LIN {X 0,Y 646.652,Z 905.532,A -85,B 0,C 180,E1 6708.912,E2 6708.912} C_VEL
LIN {X 0,Y 639.895,Z 980.734,A -85,B 0,C 180,E1 6712.285,E2 6712.285} C_VEL
LIN {X 0,Y 632.591,Z 1048.519,A -85,B 0,C 180,E1 6716.976,E2 6716.976} C_VEL
LIN {X 0,Y 626.439,Z 1105.755,A -85,B 0,C 180,E1 6722.678,E2 6722.678} C_VEL
LIN {X 0,Y 622.279,Z 1152.384,A -85,B 0,C 180,E1 6729.305,E2 6729.305} C_VEL
LIN {X 0,Y 619.924,Z 1184.854,A -85,B 0,C 180,E1 6736.2,E2 6736.2} C_VEL
LIN {X 0,Y 619.217,Z 1203.003,A -85,B 0,C 180,E1 6742.684,E2 6742.684} C_VEL
LIN {X 0,Y 619.285,Z 1209.402,A -85,B 0,C 180,E1 6747.893,E2 6747.893} C_VEL
LIN {X 0,Y 619.07,Z 1206.809,A -85,B 0,C 180,E1 6754.916,E2 6754.916} C_VEL
LIN {X 0,Y 619.272,Z 1193.72,A -85,B 0,C 180,E1 6761.152,E2 6761.152} C_VEL
LIN {X 0,Y 620.479,Z 1169.759,A -85,B 0,C 180,E1 6767.403,E2 6767.403} C_VEL
LIN {X 0,Y 623.213,Z 1133.828,A -85,B 0,C 180,E1 6773.669,E2 6773.669} C_VEL
LIN {X 0,Y 628.639,Z 1081.673,A -85,B 0,C 180,E1 6779.99,E2 6779.99} C_VEL
LIN {X 0,Y 635.999,Z 1018.12,A -85,B 0,C 180,E1 6785.354,E2 6785.354} C_VEL
LIN {X 0,Y 643.399,Z 947.885,A -85,B 0,C 180,E1 6789.377,E2 6789.377} C_VEL
LIN {X 0,Y 649.224,Z 872.681,A -85,B 0,C 180,E1 6792.052,E2 6792.052} C_VEL
LIN {X 0,Y 649.989,Z 821.956,A -85,B 0,C 180,E1 6793.177,E2 6793.177} C_VEL
LIN {X 0,Y 618.006,Z 767.06,A -85,B 0,C 180,E1 6797.097,E2 6797.097} C_VEL
LIN {X 0,Y 618.586,Z 767.06,A -85,B 0,C 180,E1 6805.206,E2 6805.206} C_VEL
LIN {X 0,Y 618.478,Z 767.06,A -85,B 0,C 180,E1 6813.498,E2 6813.498} C_VEL
LIN {X 0,Y 618.567,Z 767.06,A -85,B 0,C 180,E1 6822.165,E2 6822.165} C_VEL
LIN {X 0,Y 618.674,Z 767.06,A -85,B 0,C 180,E1 6830.844,E2 6830.844} C_VEL
LIN {X 0,Y 619.152,Z 767.06,A -85,B 0,C 180,E1 6837.908,E2 6837.908} C_VEL
LIN {X 0,Y 618.57,Z 767.06,A -85,B 0,C 180,E1 6846.859,E2 6846.859} C_VEL
LIN {X 0,Y 618.343,Z 767.06,A -85,B 0,C 180,E1 6854.941,E2 6854.941} C_VEL
LIN {X 0,Y 618.048,Z 767.06,A -85,B 0,C 180,E1 6863.063,E2 6863.063} C_VEL
LIN {X 0,Y 617.959,Z 767.06,A -85,B 0,C 180,E1 6871.87,E2 6871.87} C_VEL
LIN {X 0,Y 617.861,Z 767.06,A -85,B 0,C 180,E1 6880.604,E2 6880.604} C_VEL
LIN {X 0,Y 618.074,Z 767.06,A -85,B 0,C 180,E1 6889.157,E2 6889.157} C_VEL
LIN {X 0,Y 651.016,Z 826.368,A -85,B 0,C 180,E1 6893.12,E2 6893.12} C_VEL
LIN {X 0,Y 646.384,Z 902.657,A -85,B 0,C 180,E1 6895.132,E2 6895.132} C_VEL
LIN {X 0,Y 639.702,Z 974.081,A -85,B 0,C 180,E1 6898.439,E2 6898.439} C_VEL
LIN {X 0,Y 632.109,Z 1042.051,A -85,B 0,C 180,E1 6903.219,E2 6903.219} C_VEL
LIN {X 0,Y 625.727,Z 1100.002,A -85,B 0,C 180,E1 6909.119,E2 6909.119} C_VEL
LIN {X 0,Y 621.471,Z 1145.077,A -85,B 0,C 180,E1 6915.698,E2 6915.698} C_VEL
LIN {X 0,Y 619.614,Z 1173.985,A -85,B 0,C 180,E1 6921.912,E2 6921.912} C_VEL
LIN {X 0,Y 618.989,Z 1191.499,A -85,B 0,C 180,E1 6927.896,E2 6927.896} C_VEL
LIN {X 0,Y 619.03,Z 1199.192,A -85,B 0,C 180,E1 6933.513,E2 6933.513} C_VEL
LIN {X 0,Y 619.006,Z 1198.629,A -85,B 0,C 180,E1 6939.165,E2 6939.165} C_VEL
LIN {X 0,Y 619.22,Z 1187.747,A -85,B 0,C 180,E1 6945.63,E2 6945.63} C_VEL
LIN {X 0,Y 620.1,Z 1164.727,A -85,B 0,C 180,E1 6952.277,E2 6952.277} C_VEL
LIN {X 0,Y 622.657,Z 1130.253,A -85,B 0,C 180,E1 6958.646,E2 6958.646} C_VEL
LIN {X 0,Y 627.586,Z 1081.325,A -85,B 0,C 180,E1 6964.926,E2 6964.926} C_VEL
LIN {X 0,Y 634.691,Z 1018.951,A -85,B 0,C 180,E1 6970.528,E2 6970.528} C_VEL
LIN {X 0,Y 642.172,Z 950.633,A -85,B 0,C 180,E1 6974.718,E2 6974.718} C_VEL
LIN {X 0,Y 648.239,Z 877.127,A -85,B 0,C 180,E1 6977.607,E2 6977.607} C_VEL
LIN {X 0,Y 649.902,Z 822.371,A -85,B 0,C 180,E1 6978.954,E2 6978.954} C_VEL
LIN {X 0,Y 618.301,Z 767.06,A -85,B 0,C 180,E1 6982.858,E2 6982.858} C_VEL
LIN {X 0,Y 618.297,Z 767.06,A -85,B 0,C 180,E1 6991.404,E2 6991.404} C_VEL
LIN {X 0,Y 618.451,Z 767.06,A -85,B 0,C 180,E1 6999.152,E2 6999.152} C_VEL
LIN {X 0,Y 619.304,Z 767.06,A -85,B 0,C 180,E1 7007.969,E2 7007.969} C_VEL
LIN {X 0,Y 619.207,Z 767.06,A -85,B 0,C 180,E1 7017.88,E2 7017.88} C_VEL
LIN {X 0,Y 618.519,Z 767.06,A -85,B 0,C 180,E1 7026.786,E2 7026.786} C_VEL
LIN {X 0,Y 618.33,Z 767.06,A -85,B 0,C 180,E1 7034.912,E2 7034.912} C_VEL
LIN {X 0,Y 618.102,Z 767.06,A -85,B 0,C 180,E1 7043.065,E2 7043.065} C_VEL
LIN {X 0,Y 618.028,Z 767.06,A -85,B 0,C 180,E1 7051.833,E2 7051.833} C_VEL
LIN {X 0,Y 617.735,Z 767.06,A -85,B 0,C 180,E1 7060.577,E2 7060.577} C_VEL
LIN {X 0,Y 618.174,Z 768.815,A -85,B 0,C 180,E1 7063.107,E2 7063.107} C_VEL
LIN {X 0,Y 630.306,Z 788.536,A -85,B 0,C 180,E1 7064.58,E2 7064.58} C_VEL
LIN {X 0,Y 640.035,Z 819.345,A -85,B 0,C 180,E1 7065.934,E2 7065.934} C_VEL
LIN {X 0,Y 645.494,Z 832.84,A -85,B 0,C 180,E1 7066.641,E2 7066.641} C_VEL
LIN {X 0,Y 640.246,Z 910.482,A -85,B 0,C 180,E1 7068.61,E2 7068.61} C_VEL
LIN {X 0,Y 632.996,Z 984.571,A -85,B 0,C 180,E1 7072.046,E2 7072.046} C_VEL
LIN {X 0,Y 625.26,Z 1051.35,A -85,B 0,C 180,E1 7076.795,E2 7076.795} C_VEL
LIN {X 0,Y 618.659,Z 1108.986,A -85,B 0,C 180,E1 7082.705,E2 7082.705} C_VEL
LIN {X 0,Y 614.049,Z 1155.771,A -85,B 0,C 180,E1 7089.619,E2 7089.619} C_VEL
LIN {X 0,Y 611.637,Z 1187.515,A -85,B 0,C 180,E1 7096.74,E2 7096.74} C_VEL
LIN {X 0,Y 610.964,Z 1204.732,A -85,B 0,C 180,E1 7103.585,E2 7103.585} C_VEL
LIN {X 0,Y 610.742,Z 1209.837,A -85,B 0,C 180,E1 7109.287,E2 7109.287} C_VEL
LIN {X 0,Y 610.93,Z 1205.886,A -85,B 0,C 180,E1 7115.696,E2 7115.696} C_VEL
LIN {X 0,Y 611.296,Z 1191.049,A -85,B 0,C 180,E1 7122.171,E2 7122.171} C_VEL
LIN {X 0,Y 612.752,Z 1166.175,A -85,B 0,C 180,E1 7128.391,E2 7128.391} C_VEL
LIN {X 0,Y 616.121,Z 1128.285,A -85,B 0,C 180,E1 7134.768,E2 7134.768} C_VEL
LIN {X 0,Y 622.054,Z 1075.538,A -85,B 0,C 180,E1 7140.989,E2 7140.989} C_VEL
LIN {X 0,Y 629.962,Z 1011.452,A -85,B 0,C 180,E1 7146.255,E2 7146.255} C_VEL
LIN {X 0,Y 637.699,Z 941.735,A -85,B 0,C 180,E1 7150.117,E2 7150.117} C_VEL
LIN {X 0,Y 643.46,Z 869.863,A -85,B 0,C 180,E1 7152.597,E2 7152.597} C_VEL
LIN {X 0,Y 644.183,Z 825.386,A -85,B 0,C 180,E1 7153.602,E2 7153.602} C_VEL
LIN {X 0,Y 610.109,Z 767.06,A -85,B 0,C 180,E1 7157.757,E2 7157.757} C_VEL
LIN {X 0,Y 610.507,Z 767.06,A -85,B 0,C 180,E1 7166.313,E2 7166.313} C_VEL
LIN {X 0,Y 610.224,Z 767.06,A -85,B 0,C 180,E1 7175.097,E2 7175.097} C_VEL
LIN {X 0,Y 610.432,Z 767.06,A -85,B 0,C 180,E1 7183.41,E2 7183.41} C_VEL
LIN {X 0,Y 610.395,Z 767.06,A -85,B 0,C 180,E1 7192.159,E2 7192.159} C_VEL
LIN {X 0,Y 610.543,Z 767.06,A -85,B 0,C 180,E1 7199.302,E2 7199.302} C_VEL
LIN {X 0,Y 610.719,Z 767.06,A -85,B 0,C 180,E1 7206.432,E2 7206.432} C_VEL
LIN {X 0,Y 610.288,Z 767.06,A -85,B 0,C 180,E1 7215.143,E2 7215.143} C_VEL
LIN {X 0,Y 610.126,Z 767.06,A -85,B 0,C 180,E1 7222.681,E2 7222.681} C_VEL
LIN {X 0,Y 610.031,Z 767.06,A -85,B 0,C 180,E1 7230.953,E2 7230.953} C_VEL
LIN {X 0,Y 609.928,Z 767.06,A -85,B 0,C 180,E1 7239.377,E2 7239.377} C_VEL
LIN {X 0,Y 610.104,Z 767.06,A -85,B 0,C 180,E1 7248.363,E2 7248.363} C_VEL
LIN {X 0,Y 644.99,Z 830.304,A -85,B 0,C 180,E1 7252.71,E2 7252.71} C_VEL
LIN {X 0,Y 640.023,Z 905.813,A -85,B 0,C 180,E1 7254.768,E2 7254.768} C_VEL
LIN {X 0,Y 632.651,Z 978.92,A -85,B 0,C 180,E1 7258.259,E2 7258.259} C_VEL
LIN {X 0,Y 624.558,Z 1046.254,A -85,B 0,C 180,E1 7263.167,E2 7263.167} C_VEL
LIN {X 0,Y 617.852,Z 1103.053,A -85,B 0,C 180,E1 7269.154,E2 7269.154} C_VEL
LIN {X 0,Y 613.555,Z 1146.482,A -85,B 0,C 180,E1 7275.693,E2 7275.693} C_VEL
LIN {X 0,Y 611.53,Z 1175.593,A -85,B 0,C 180,E1 7282.163,E2 7282.163} C_VEL
LIN {X 0,Y 610.998,Z 1191.666,A -85,B 0,C 180,E1 7287.868,E2 7287.868} C_VEL
LIN {X 0,Y 611.032,Z 1199.245,A -85,B 0,C 180,E1 7293.559,E2 7293.559} C_VEL
LIN {X 0,Y 610.978,Z 1198.565,A -85,B 0,C 180,E1 7299.286,E2 7299.286} C_VEL
LIN {X 0,Y 611.202,Z 1187.536,A -85,B 0,C 180,E1 7305.84,E2 7305.84} C_VEL
LIN {X 0,Y 612.166,Z 1165.432,A -85,B 0,C 180,E1 7312.328,E2 7312.328} C_VEL
LIN {X 0,Y 614.89,Z 1130.949,A -85,B 0,C 180,E1 7318.838,E2 7318.838} C_VEL
LIN {X 0,Y 620.221,Z 1081.784,A -85,B 0,C 180,E1 7325.251,E2 7325.251} C_VEL
LIN {X 0,Y 627.846,Z 1019.141,A -85,B 0,C 180,E1 7330.943,E2 7330.943} C_VEL
LIN {X 0,Y 635.752,Z 950.839,A -85,B 0,C 180,E1 7335.172,E2 7335.172} C_VEL
LIN {X 0,Y 642.175,Z 877.876,A -85,B 0,C 180,E1 7338.064,E2 7338.064} C_VEL
LIN {X 0,Y 643.929,Z 825.752,A -85,B 0,C 180,E1 7339.389,E2 7339.389} C_VEL
LIN {X 0,Y 610.217,Z 767.06,A -85,B 0,C 180,E1 7343.569,E2 7343.569} C_VEL
LIN {X 0,Y 610.195,Z 767.06,A -85,B 0,C 180,E1 7352.604,E2 7352.604} C_VEL
LIN {X 0,Y 610.314,Z 767.06,A -85,B 0,C 180,E1 7360.38,E2 7360.38} C_VEL
LIN {X 0,Y 611.208,Z 767.06,A -85,B 0,C 180,E1 7369.258,E2 7369.258} C_VEL
LIN {X 0,Y 611.225,Z 767.06,A -85,B 0,C 180,E1 7377.852,E2 7377.852} C_VEL
LIN {X 0,Y 610.649,Z 767.06,A -85,B 0,C 180,E1 7386.404,E2 7386.404} C_VEL
LIN {X 0,Y 610.277,Z 767.06,A -85,B 0,C 180,E1 7395.113,E2 7395.113} C_VEL
LIN {X 0,Y 610.171,Z 767.06,A -85,B 0,C 180,E1 7402.648,E2 7402.648} C_VEL
LIN {X 0,Y 610.093,Z 767.06,A -85,B 0,C 180,E1 7410.955,E2 7410.955} C_VEL
LIN {X 0,Y 609.826,Z 767.06,A -85,B 0,C 180,E1 7419.348,E2 7419.348} C_VEL
LIN {X 0,Y 609.968,Z 768.528,A -85,B 0,C 180,E1 7422.277,E2 7422.277} C_VEL
LIN {X 0,Y 640.035,Z 819.345,A -85,B 0,C 180,E1 7425.934,E2 7425.934} C_VEL
LIN {X 0,Y 641.851,Z 835.895,A -85,B 0,C 180,E1 7426.391,E2 7426.391} C_VEL
LIN {X 0,Y 638.694,Z 854.619,A -85,B 0,C 180,E1 7426.566,E2 7426.566} C_VEL
LIN {X 0,Y 632.966,Z 925.708,A -85,B 0,C 180,E1 7428.72,E2 7428.72} C_VEL
LIN {X 0,Y 624.969,Z 998.18,A -85,B 0,C 180,E1 7432.423,E2 7432.423} C_VEL
LIN {X 0,Y 616.681,Z 1063.626,A -85,B 0,C 180,E1 7437.476,E2 7437.476} C_VEL
LIN {X 0,Y 609.86,Z 1118.897,A -85,B 0,C 180,E1 7443.617,E2 7443.617} C_VEL
LIN {X 0,Y 605.354,Z 1162.455,A -85,B 0,C 180,E1 7450.612,E2 7450.612} C_VEL
LIN {X 0,Y 603.417,Z 1189.883,A -85,B 0,C 180,E1 7457.295,E2 7457.295} C_VEL
LIN {X 0,Y 602.986,Z 1204.729,A -85,B 0,C 180,E1 7463.5,E2 7463.5} C_VEL
LIN {X 0,Y 602.743,Z 1209.837,A -85,B 0,C 180,E1 7469.277,E2 7469.277} C_VEL
LIN {X 0,Y 602.939,Z 1205.886,A -85,B 0,C 180,E1 7475.772,E2 7475.772} C_VEL
LIN {X 0,Y 603.33,Z 1191.046,A -85,B 0,C 180,E1 7482.334,E2 7482.334} C_VEL
LIN {X 0,Y 604.898,Z 1166.177,A -85,B 0,C 180,E1 7488.639,E2 7488.639} C_VEL
LIN {X 0,Y 608.667,Z 1127.165,A -85,B 0,C 180,E1 7495.258,E2 7495.258} C_VEL
LIN {X 0,Y 615.193,Z 1073.255,A -85,B 0,C 180,E1 7501.619,E2 7501.619} C_VEL
LIN {X 0,Y 623.552,Z 1009.569,A -85,B 0,C 180,E1 7506.835,E2 7506.835} C_VEL
LIN {X 0,Y 631.629,Z 940.402,A -85,B 0,C 180,E1 7510.653,E2 7510.653} C_VEL
LIN {X 0,Y 637.635,Z 868.9,A -85,B 0,C 180,E1 7513.108,E2 7513.108} C_VEL
LIN {X 0,Y 638.249,Z 828.483,A -85,B 0,C 180,E1 7514.054,E2 7514.054} C_VEL
LIN {X 0,Y 602.17,Z 767.06,A -85,B 0,C 180,E1 7518.662,E2 7518.662} C_VEL
LIN {X 0,Y 602.419,Z 767.06,A -85,B 0,C 180,E1 7527.485,E2 7527.485} C_VEL
LIN {X 0,Y 602.185,Z 767.06,A -85,B 0,C 180,E1 7535.457,E2 7535.457} C_VEL
LIN {X 0,Y 602.46,Z 767.06,A -85,B 0,C 180,E1 7543.184,E2 7543.184} C_VEL
LIN {X 0,Y 602.432,Z 767.06,A -85,B 0,C 180,E1 7552.054,E2 7552.054} C_VEL
LIN {X 0,Y 602.544,Z 767.06,A -85,B 0,C 180,E1 7559.293,E2 7559.293} C_VEL
LIN {X 0,Y 602.705,Z 767.06,A -85,B 0,C 180,E1 7566.517,E2 7566.517} C_VEL
LIN {X 0,Y 602.244,Z 767.06,A -85,B 0,C 180,E1 7575.35,E2 7575.35} C_VEL
LIN {X 0,Y 602.017,Z 767.06,A -85,B 0,C 180,E1 7583.164,E2 7583.164} C_VEL
LIN {X 0,Y 602.026,Z 767.06,A -85,B 0,C 180,E1 7591.116,E2 7591.116} C_VEL
LIN {X 0,Y 601.862,Z 767.06,A -85,B 0,C 180,E1 7600.01,E2 7600.01} C_VEL
LIN {X 0,Y 602.326,Z 768.684,A -85,B 0,C 180,E1 7607.588,E2 7607.588} C_VEL
LIN {X 0,Y 639.071,Z 831.669,A -85,B 0,C 180,E1 7612.243,E2 7612.243} C_VEL
LIN {X 0,Y 633.792,Z 906.945,A -85,B 0,C 180,E1 7614.327,E2 7614.327} C_VEL
LIN {X 0,Y 626.144,Z 978.79,A -85,B 0,C 180,E1 7617.788,E2 7617.788} C_VEL
LIN {X 0,Y 617.555,Z 1046.251,A -85,B 0,C 180,E1 7622.747,E2 7622.747} C_VEL
LIN {X 0,Y 610.312,Z 1103.709,A -85,B 0,C 180,E1 7628.884,E2 7628.884} C_VEL
LIN {X 0,Y 605.742,Z 1146.922,A -85,B 0,C 180,E1 7635.504,E2 7635.504} C_VEL
LIN {X 0,Y 603.583,Z 1175.885,A -85,B 0,C 180,E1 7642.059,E2 7642.059} C_VEL
LIN {X 0,Y 603.006,Z 1191.828,A -85,B 0,C 180,E1 7647.84,E2 7647.84} C_VEL
LIN {X 0,Y 603.013,Z 1199.293,A -85,B 0,C 180,E1 7653.607,E2 7653.607} C_VEL
LIN {X 0,Y 602.959,Z 1198.499,A -85,B 0,C 180,E1 7659.411,E2 7659.411} C_VEL
LIN {X 0,Y 603.201,Z 1187.324,A -85,B 0,C 180,E1 7666.056,E2 7666.056} C_VEL
LIN {X 0,Y 604.221,Z 1165.961,A -85,B 0,C 180,E1 7672.422,E2 7672.422} C_VEL
LIN {X 0,Y 607.089,Z 1132.198,A -85,B 0,C 180,E1 7678.946,E2 7678.946} C_VEL
LIN {X 0,Y 612.799,Z 1082.461,A -85,B 0,C 180,E1 7685.561,E2 7685.561} C_VEL
LIN {X 0,Y 620.822,Z 1020.755,A -85,B 0,C 180,E1 7691.261,E2 7691.261} C_VEL
LIN {X 0,Y 629.244,Z 952.328,A -85,B 0,C 180,E1 7695.569,E2 7695.569} C_VEL
LIN {X 0,Y 636.186,Z 878.289,A -85,B 0,C 180,E1 7698.538,E2 7698.538} C_VEL
LIN {X 0,Y 637.97,Z 829.221,A -85,B 0,C 180,E1 7699.822,E2 7699.822} C_VEL
LIN {X 0,Y 602.129,Z 767.06,A -85,B 0,C 180,E1 7704.51,E2 7704.51} C_VEL
LIN {X 0,Y 602.148,Z 767.06,A -85,B 0,C 180,E1 7713.39,E2 7713.39} C_VEL
LIN {X 0,Y 602.295,Z 767.06,A -85,B 0,C 180,E1 7721.636,E2 7721.636} C_VEL
LIN {X 0,Y 603.232,Z 767.06,A -85,B 0,C 180,E1 7729.115,E2 7729.115} C_VEL
LIN {X 0,Y 603.222,Z 767.06,A -85,B 0,C 180,E1 7737.824,E2 7737.824} C_VEL
LIN {X 0,Y 602.619,Z 767.06,A -85,B 0,C 180,E1 7746.489,E2 7746.489} C_VEL
LIN {X 0,Y 602.232,Z 767.06,A -85,B 0,C 180,E1 7755.32,E2 7755.32} C_VEL
LIN {X 0,Y 602.087,Z 767.06,A -85,B 0,C 180,E1 7763.169,E2 7763.169} C_VEL
LIN {X 0,Y 602.088,Z 767.06,A -85,B 0,C 180,E1 7771.078,E2 7771.078} C_VEL
LIN {X 0,Y 601.745,Z 767.06,A -85,B 0,C 180,E1 7779.982,E2 7779.982} C_VEL
LIN {X 0,Y 602.006,Z 769.142,A -85,B 0,C 180,E1 7781.44,E2 7781.44} C_VEL
LIN {X 0,Y 638.942,Z 831.754,A -85,B 0,C 180,E1 7786.065,E2 7786.065} C_VEL
LIN {X 0,Y 638.694,Z 854.619,A -85,B 0,C 180,E1 7786.566,E2 7786.566} C_VEL
LIN {X 0,Y 630.175,Z 888.867,A -85,B 0,C 180,E1 7786.933,E2 7786.933} C_VEL
LIN {X 0,Y 622.818,Z 963.473,A -85,B 0,C 180,E1 7789.963,E2 7789.963} C_VEL
LIN {X 0,Y 613.767,Z 1032.869,A -85,B 0,C 180,E1 7794.408,E2 7794.408} C_VEL
LIN {X 0,Y 605.285,Z 1094.461,A -85,B 0,C 180,E1 7800.225,E2 7800.225} C_VEL
LIN {X 0,Y 599.44,Z 1144.557,A -85,B 0,C 180,E1 7807.084,E2 7807.084} C_VEL
LIN {X 0,Y 596.577,Z 1180.801,A -85,B 0,C 180,E1 7814.518,E2 7814.518} C_VEL
LIN {X 0,Y 595.461,Z 1202.16,A -85,B 0,C 180,E1 7821.946,E2 7821.946} C_VEL
LIN {X 0,Y 595.295,Z 1209.402,A -85,B 0,C 180,E1 7827.808,E2 7827.808} C_VEL
LIN {X 0,Y 595.057,Z 1206.8,A -85,B 0,C 180,E1 7835.115,E2 7835.115} C_VEL
LIN {X 0,Y 595.284,Z 1193.106,A -85,B 0,C 180,E1 7841.823,E2 7841.823} C_VEL
LIN {X 0,Y 596.865,Z 1169.068,A -85,B 0,C 180,E1 7848.266,E2 7848.266} C_VEL
LIN {X 0,Y 600.631,Z 1131.177,A -85,B 0,C 180,E1 7855.015,E2 7855.015} C_VEL
LIN {X 0,Y 607.245,Z 1079.171,A -85,B 0,C 180,E1 7861.434,E2 7861.434} C_VEL
LIN {X 0,Y 616.093,Z 1015.607,A -85,B 0,C 180,E1 7866.877,E2 7866.877} C_VEL
LIN {X 0,Y 624.756,Z 946.468,A -85,B 0,C 180,E1 7870.87,E2 7870.87} C_VEL
LIN {X 0,Y 631.517,Z 872.325,A -85,B 0,C 180,E1 7873.527,E2 7873.527} C_VEL
LIN {X 0,Y 632.417,Z 831.751,A -85,B 0,C 180,E1 7874.505,E2 7874.505} C_VEL
LIN {X 0,Y 594.256,Z 767.06,A -85,B 0,C 180,E1 7879.644,E2 7879.644} C_VEL
LIN {X 0,Y 594.349,Z 767.06,A -85,B 0,C 180,E1 7888.727,E2 7888.727} C_VEL
LIN {X 0,Y 594.042,Z 767.06,A -85,B 0,C 180,E1 7896.701,E2 7896.701} C_VEL
LIN {X 0,Y 594.244,Z 767.06,A -85,B 0,C 180,E1 7904.469,E2 7904.469} C_VEL
LIN {X 0,Y 594.437,Z 767.06,A -85,B 0,C 180,E1 7911.947,E2 7911.947} C_VEL
LIN {X 0,Y 594.556,Z 767.06,A -85,B 0,C 180,E1 7919.284,E2 7919.284} C_VEL
LIN {X 0,Y 594.669,Z 767.06,A -85,B 0,C 180,E1 7926.606,E2 7926.606} C_VEL
LIN {X 0,Y 594.204,Z 767.06,A -85,B 0,C 180,E1 7935.563,E2 7935.563} C_VEL
LIN {X 0,Y 593.993,Z 767.06,A -85,B 0,C 180,E1 7943.333,E2 7943.333} C_VEL
LIN {X 0,Y 593.973,Z 767.06,A -85,B 0,C 180,E1 7951.586,E2 7951.586} C_VEL
LIN {X 0,Y 593.795,Z 767.06,A -85,B 0,C 180,E1 7960.667,E2 7960.667} C_VEL
LIN {X 0,Y 594.414,Z 769.008,A -85,B 0,C 180,E1 7966.746,E2 7966.746} C_VEL
LIN {X 0,Y 633.123,Z 835.281,A -85,B 0,C 180,E1 7971.815,E2 7971.815} C_VEL
LIN {X 0,Y 627.447,Z 909.958,A -85,B 0,C 180,E1 7973.955,E2 7973.955} C_VEL
LIN {X 0,Y 619.222,Z 981.916,A -85,B 0,C 180,E1 7977.511,E2 7977.511} C_VEL
LIN {X 0,Y 610.248,Z 1048.399,A -85,B 0,C 180,E1 7982.516,E2 7982.516} C_VEL
LIN {X 0,Y 602.561,Z 1105.875,A -85,B 0,C 180,E1 7988.808,E2 7988.808} C_VEL
LIN {X 0,Y 597.692,Z 1149.281,A -85,B 0,C 180,E1 7995.68,E2 7995.68} C_VEL
LIN {X 0,Y 595.53,Z 1177.485,A -85,B 0,C 180,E1 8002.319,E2 8002.319} C_VEL
LIN {X 0,Y 594.889,Z 1193.365,A -85,B 0,C 180,E1 8008.541,E2 8008.541} C_VEL
LIN {X 0,Y 595.007,Z 1199.34,A -85,B 0,C 180,E1 8013.655,E2 8013.655} C_VEL
LIN {X 0,Y 594.885,Z 1196.995,A -85,B 0,C 180,E1 8020.906,E2 8020.906} C_VEL
LIN {X 0,Y 595.419,Z 1183.037,A -85,B 0,C 180,E1 8027.797,E2 8027.797} C_VEL
LIN {X 0,Y 597.458,Z 1155.363,A -85,B 0,C 180,E1 8035.014,E2 8035.014} C_VEL
LIN {X 0,Y 601.902,Z 1113.172,A -85,B 0,C 180,E1 8042.115,E2 8042.115} C_VEL
LIN {X 0,Y 608.914,Z 1058.814,A -85,B 0,C 180,E1 8048.421,E2 8048.421} C_VEL
LIN {X 0,Y 617.715,Z 993.256,A -85,B 0,C 180,E1 8053.681,E2 8053.681} C_VEL
LIN {X 0,Y 626.349,Z 921.171,A -85,B 0,C 180,E1 8057.505,E2 8057.505} C_VEL
LIN {X 0,Y 632.508,Z 850.17,A -85,B 0,C 180,E1 8059.764,E2 8059.764} C_VEL
LIN {X 0,Y 631.637,Z 831.834,A -85,B 0,C 180,E1 8060.312,E2 8060.312} C_VEL
LIN {X 0,Y 594.082,Z 767.06,A -85,B 0,C 180,E1 8065.523,E2 8065.523} C_VEL
LIN {X 0,Y 594.155,Z 767.06,A -85,B 0,C 180,E1 8073.447,E2 8073.447} C_VEL
LIN {X 0,Y 594.3,Z 767.06,A -85,B 0,C 180,E1 8081.38,E2 8081.38} C_VEL
LIN {X 0,Y 595.216,Z 767.06,A -85,B 0,C 180,E1 8088.966,E2 8088.966} C_VEL
LIN {X 0,Y 595.217,Z 767.06,A -85,B 0,C 180,E1 8097.795,E2 8097.795} C_VEL
LIN {X 0,Y 594.584,Z 767.06,A -85,B 0,C 180,E1 8106.577,E2 8106.577} C_VEL
LIN {X 0,Y 594.191,Z 767.06,A -85,B 0,C 180,E1 8115.533,E2 8115.533} C_VEL
LIN {X 0,Y 594.066,Z 767.06,A -85,B 0,C 180,E1 8123.298,E2 8123.298} C_VEL
LIN {X 0,Y 594.04,Z 767.06,A -85,B 0,C 180,E1 8131.547,E2 8131.547} C_VEL
LIN {X 0,Y 593.742,Z 767.575,A -85,B 0,C 180,E1 8140.469,E2 8140.469} C_VEL
LIN {X 0,Y 633.662,Z 836.021,A -85,B 0,C 180,E1 8145.685,E2 8145.685} C_VEL
LIN {X 0,Y 630.175,Z 888.867,A -85,B 0,C 180,E1 8146.933,E2 8146.933} C_VEL
LIN {X 0,Y 622.012,Z 911.312,A -85,B 0,C 180,E1 8147.149,E2 8147.149} C_VEL
LIN {X 0,Y 613.5,Z 985.783,A -85,B 0,C 180,E1 8150.693,E2 8150.693} C_VEL
LIN {X 0,Y 604.267,Z 1052.795,A -85,B 0,C 180,E1 8155.619,E2 8155.619} C_VEL
LIN {X 0,Y 596.167,Z 1110.284,A -85,B 0,C 180,E1 8161.755,E2 8161.755} C_VEL
LIN {X 0,Y 590.789,Z 1156.571,A -85,B 0,C 180,E1 8168.937,E2 8168.937} C_VEL
LIN {X 0,Y 587.778,Z 1188.725,A -85,B 0,C 180,E1 8176.571,E2 8176.571} C_VEL
LIN {X 0,Y 587.05,Z 1204.724,A -85,B 0,C 180,E1 8183.323,E2 8183.323} C_VEL
LIN {X 0,Y 586.748,Z 1209.837,A -85,B 0,C 180,E1 8189.257,E2 8189.257} C_VEL
LIN {X 0,Y 586.952,Z 1205.919,A -85,B 0,C 180,E1 8195.904,E2 8195.904} C_VEL
LIN {X 0,Y 587.436,Z 1191.04,A -85,B 0,C 180,E1 8202.673,E2 8202.673} C_VEL
LIN {X 0,Y 589.496,Z 1164.51,A -85,B 0,C 180,E1 8209.514,E2 8209.514} C_VEL
LIN {X 0,Y 594.465,Z 1121.523,A -85,B 0,C 180,E1 8216.753,E2 8216.753} C_VEL
LIN {X 0,Y 602.099,Z 1066.601,A -85,B 0,C 180,E1 8223.108,E2 8223.108} C_VEL
LIN {X 0,Y 611.544,Z 1001.134,A -85,B 0,C 180,E1 8228.334,E2 8228.334} C_VEL
LIN {X 0,Y 620.461,Z 929.695,A -85,B 0,C 180,E1 8232.108,E2 8232.108} C_VEL
LIN {X 0,Y 626.59,Z 860.944,A -85,B 0,C 180,E1 8234.299,E2 8234.299} C_VEL
LIN {X 0,Y 626.419,Z 834.814,A -85,B 0,C 180,E1 8234.986,E2 8234.986} C_VEL
LIN {X 0,Y 586.263,Z 767.06,A -85,B 0,C 180,E1 8240.464,E2 8240.464} C_VEL
LIN {X 0,Y 586.296,Z 767.06,A -85,B 0,C 180,E1 8247.987,E2 8247.987} C_VEL
LIN {X 0,Y 586.04,Z 767.06,A -85,B 0,C 180,E1 8256.718,E2 8256.718} C_VEL
LIN {X 0,Y 586.253,Z 767.06,A -85,B 0,C 180,E1 8264.251,E2 8264.251} C_VEL
LIN {X 0,Y 586.452,Z 767.06,A -85,B 0,C 180,E1 8271.836,E2 8271.836} C_VEL
LIN {X 0,Y 586.557,Z 767.06,A -85,B 0,C 180,E1 8279.274,E2 8279.274} C_VEL
LIN {X 0,Y 586.637,Z 767.06,A -85,B 0,C 180,E1 8286.697,E2 8286.697} C_VEL
LIN {X 0,Y 586.454,Z 767.06,A -85,B 0,C 180,E1 8294.239,E2 8294.239} C_VEL
LIN {X 0,Y 585.994,Z 767.06,A -85,B 0,C 180,E1 8303.271,E2 8303.271} C_VEL
LIN {X 0,Y 585.886,Z 767.06,A -85,B 0,C 180,E1 8312.073,E2 8312.073} C_VEL
LIN {X 0,Y 585.798,Z 767.06,A -85,B 0,C 180,E1 8321.342,E2 8321.342} C_VEL
LIN {X 0,Y 586.257,Z 768.601,A -85,B 0,C 180,E1 8325.839,E2 8325.839} C_VEL
LIN {X 0,Y 627.142,Z 837.925,A -85,B 0,C 180,E1 8331.348,E2 8331.348} C_VEL
LIN {X 0,Y 621.227,Z 911.888,A -85,B 0,C 180,E1 8333.531,E2 8333.531} C_VEL
LIN {X 0,Y 612.575,Z 983.23,A -85,B 0,C 180,E1 8337.114,E2 8337.114} C_VEL
LIN {X 0,Y 603.245,Z 1048.719,A -85,B 0,C 180,E1 8342.108,E2 8342.108} C_VEL
LIN {X 0,Y 595.295,Z 1104.999,A -85,B 0,C 180,E1 8348.325,E2 8348.325} C_VEL
LIN {X 0,Y 590.12,Z 1147.905,A -85,B 0,C 180,E1 8355.132,E2 8355.132} C_VEL
LIN {X 0,Y 587.584,Z 1177.753,A -85,B 0,C 180,E1 8362.215,E2 8362.215} C_VEL
LIN {X 0,Y 586.9,Z 1193.501,A -85,B 0,C 180,E1 8368.522,E2 8368.522} C_VEL
LIN {X 0,Y 586.989,Z 1199.387,A -85,B 0,C 180,E1 8373.705,E2 8373.705} C_VEL
LIN {X 0,Y 586.947,Z 1198.365,A -85,B 0,C 180,E1 8379.67,E2 8379.67} C_VEL
LIN {X 0,Y 587.219,Z 1186.952,A -85,B 0,C 180,E1 8386.477,E2 8386.477} C_VEL
LIN {X 0,Y 588.531,Z 1164.891,A -85,B 0,C 180,E1 8393.14,E2 8393.14} C_VEL
LIN {X 0,Y 591.914,Z 1129.776,A -85,B 0,C 180,E1 8399.975,E2 8399.975} C_VEL
LIN {X 0,Y 598.67,Z 1079.518,A -85,B 0,C 180,E1 8406.687,E2 8406.687} C_VEL
LIN {X 0,Y 607.793,Z 1017.294,A -85,B 0,C 180,E1 8412.44,E2 8412.44} C_VEL
LIN {X 0,Y 617.109,Z 949.117,A -85,B 0,C 180,E1 8416.705,E2 8416.705} C_VEL
LIN {X 0,Y 624.477,Z 877.987,A -85,B 0,C 180,E1 8419.545,E2 8419.545} C_VEL
LIN {X 0,Y 626.048,Z 835.954,A -85,B 0,C 180,E1 8420.711,E2 8420.711} C_VEL
LIN {X 0,Y 588.518,Z 772.778,A -85,B 0,C 180,E1 8425.856,E2 8425.856} C_VEL
LIN {X 0,Y 586.079,Z 767.06,A -85,B 0,C 180,E1 8426.456,E2 8426.456} C_VEL
LIN {X 0,Y 586.196,Z 767.06,A -85,B 0,C 180,E1 8434.709,E2 8434.709} C_VEL
LIN {X 0,Y 586.682,Z 767.06,A -85,B 0,C 180,E1 8444.233,E2 8444.233} C_VEL
LIN {X 0,Y 586.54,Z 767.06,A -85,B 0,C 180,E1 8451.808,E2 8451.808} C_VEL
LIN {X 0,Y 586.591,Z 767.06,A -85,B 0,C 180,E1 8459.244,E2 8459.244} C_VEL
LIN {X 0,Y 586.571,Z 767.06,A -85,B 0,C 180,E1 8466.668,E2 8466.668} C_VEL
LIN {X 0,Y 586.457,Z 767.06,A -85,B 0,C 180,E1 8474.209,E2 8474.209} C_VEL
LIN {X 0,Y 586.07,Z 767.06,A -85,B 0,C 180,E1 8483.278,E2 8483.278} C_VEL
LIN {X 0,Y 585.95,Z 767.06,A -85,B 0,C 180,E1 8492.034,E2 8492.034} C_VEL
LIN {X 0,Y 585.991,Z 768.878,A -85,B 0,C 180,E1 8499.556,E2 8499.556} C_VEL
LIN {X 0,Y 622.905,Z 829.875,A -85,B 0,C 180,E1 8504.599,E2 8504.599} C_VEL
LIN {X 0,Y 627.63,Z 844.106,A -85,B 0,C 180,E1 8505.348,E2 8505.348} C_VEL
LIN {X 0,Y 622.012,Z 911.312,A -85,B 0,C 180,E1 8507.149,E2 8507.149} C_VEL
LIN {X 0,Y 612.707,Z 944.277,A -85,B 0,C 180,E1 8508.027,E2 8508.027} C_VEL
LIN {X 0,Y 603.123,Z 1014.101,A -85,B 0,C 180,E1 8512.071,E2 8512.071} C_VEL
LIN {X 0,Y 593.151,Z 1078.693,A -85,B 0,C 180,E1 8517.676,E2 8517.676} C_VEL
LIN {X 0,Y 585.628,Z 1131.143,A -85,B 0,C 180,E1 8524.293,E2 8524.293} C_VEL
LIN {X 0,Y 581.338,Z 1167.92,A -85,B 0,C 180,E1 8530.967,E2 8530.967} C_VEL
LIN {X 0,Y 579.286,Z 1193.288,A -85,B 0,C 180,E1 8537.909,E2 8537.909} C_VEL
LIN {X 0,Y 578.968,Z 1206.789,A -85,B 0,C 180,E1 8544.738,E2 8544.738} C_VEL
LIN {X 0,Y 578.637,Z 1209.838,A -85,B 0,C 180,E1 8550.749,E2 8550.749} C_VEL
LIN {X 0,Y 579.203,Z 1203.517,A -85,B 0,C 180,E1 8557.52,E2 8557.52} C_VEL
LIN {X 0,Y 580.551,Z 1183.675,A -85,B 0,C 180,E1 8565.097,E2 8565.097} C_VEL
LIN {X 0,Y 583.682,Z 1148.476,A -85,B 0,C 180,E1 8572.855,E2 8572.855} C_VEL
LIN {X 0,Y 589.96,Z 1100.701,A -85,B 0,C 180,E1 8579.834,E2 8579.834} C_VEL
LIN {X 0,Y 599.01,Z 1041.871,A -85,B 0,C 180,E1 8585.778,E2 8585.778} C_VEL
LIN {X 0,Y 608.877,Z 973.421,A -85,B 0,C 180,E1 8590.508,E2 8590.508} C_VEL
LIN {X 0,Y 617.236,Z 899.379,A -85,B 0,C 180,E1 8593.774,E2 8593.774} C_VEL
LIN {X 0,Y 620.679,Z 838.301,A -85,B 0,C 180,E1 8595.431,E2 8595.431} C_VEL
LIN {X 0,Y 578.248,Z 767.06,A -85,B 0,C 180,E1 8601.453,E2 8601.453} C_VEL
LIN {X 0,Y 578.248,Z 767.06,A -85,B 0,C 180,E1 8609.252,E2 8609.252} C_VEL
LIN {X 0,Y 578.069,Z 767.06,A -85,B 0,C 180,E1 8618.629,E2 8618.629} C_VEL
LIN {X 0,Y 578.386,Z 767.06,A -85,B 0,C 180,E1 8627.135,E2 8627.135} C_VEL
LIN {X 0,Y 579.023,Z 767.06,A -85,B 0,C 180,E1 8636.26,E2 8636.26} C_VEL
LIN {X 0,Y 579.048,Z 767.06,A -85,B 0,C 180,E1 8645.276,E2 8645.276} C_VEL
LIN {X 0,Y 578.392,Z 767.06,A -85,B 0,C 180,E1 8654.442,E2 8654.442} C_VEL
LIN {X 0,Y 578.065,Z 767.06,A -85,B 0,C 180,E1 8662.38,E2 8662.38} C_VEL
LIN {X 0,Y 577.883,Z 767.06,A -85,B 0,C 180,E1 8671.481,E2 8671.481} C_VEL
LIN {X 0,Y 577.761,Z 767.06,A -85,B 0,C 180,E1 8680.052,E2 8680.052} C_VEL
LIN {X 0,Y 578.298,Z 769.023,A -85,B 0,C 180,E1 8684.937,E2 8684.937} C_VEL
LIN {X 0,Y 620.36,Z 839.379,A -85,B 0,C 180,E1 8690.763,E2 8690.763} C_VEL
LIN {X 0,Y 614.724,Z 917.092,A -85,B 0,C 180,E1 8693.233,E2 8693.233} C_VEL
LIN {X 0,Y 605.555,Z 987.423,A -85,B 0,C 180,E1 8696.894,E2 8696.894} C_VEL
LIN {X 0,Y 595.549,Z 1053.428,A -85,B 0,C 180,E1 8702.105,E2 8702.105} C_VEL
LIN {X 0,Y 587.15,Z 1109.675,A -85,B 0,C 180,E1 8708.58,E2 8708.58} C_VEL
LIN {X 0,Y 581.832,Z 1152.033,A -85,B 0,C 180,E1 8715.666,E2 8715.666} C_VEL
LIN {X 0,Y 579.532,Z 1179.184,A -85,B 0,C 180,E1 8722.484,E2 8722.484} C_VEL
LIN {X 0,Y 578.923,Z 1193.63,A -85,B 0,C 180,E1 8728.501,E2 8728.501} C_VEL
LIN {X 0,Y 578.988,Z 1199.434,A -85,B 0,C 180,E1 8733.757,E2 8733.757} C_VEL
LIN {X 0,Y 578.958,Z 1196.659,A -85,B 0,C 180,E1 8741.331,E2 8741.331} C_VEL
LIN {X 0,Y 579.838,Z 1181.361,A -85,B 0,C 180,E1 8748.688,E2 8748.688} C_VEL
LIN {X 0,Y 582.65,Z 1150.74,A -85,B 0,C 180,E1 8756.479,E2 8756.479} C_VEL
LIN {X 0,Y 587.827,Z 1106.927,A -85,B 0,C 180,E1 8763.689,E2 8763.689} C_VEL
LIN {X 0,Y 596.085,Z 1050.675,A -85,B 0,C 180,E1 8770.059,E2 8770.059} C_VEL
LIN {X 0,Y 605.808,Z 984.65,A -85,B 0,C 180,E1 8775.206,E2 8775.206} C_VEL
LIN {X 0,Y 615.259,Z 910.684,A -85,B 0,C 180,E1 8778.951,E2 8778.951} C_VEL
LIN {X 0,Y 620.213,Z 839.378,A -85,B 0,C 180,E1 8781.162,E2 8781.162} C_VEL
LIN {X 0,Y 584.495,Z 778.715,A -85,B 0,C 180,E1 8786.237,E2 8786.237} C_VEL
LIN {X 0,Y 578.097,Z 767.06,A -85,B 0,C 180,E1 8787.442,E2 8787.442} C_VEL
LIN {X 0,Y 578.264,Z 767.06,A -85,B 0,C 180,E1 8795.993,E2 8795.993} C_VEL
LIN {X 0,Y 578.938,Z 767.06,A -85,B 0,C 180,E1 8805.572,E2 8805.572} C_VEL
LIN {X 0,Y 578.356,Z 767.06,A -85,B 0,C 180,E1 8813.207,E2 8813.207} C_VEL
LIN {X 0,Y 578.615,Z 767.06,A -85,B 0,C 180,E1 8819.234,E2 8819.234} C_VEL
LIN {X 0,Y 578.536,Z 767.06,A -85,B 0,C 180,E1 8826.761,E2 8826.761} C_VEL
LIN {X 0,Y 578.392,Z 767.06,A -85,B 0,C 180,E1 8834.411,E2 8834.411} C_VEL
LIN {X 0,Y 578.159,Z 767.06,A -85,B 0,C 180,E1 8842.344,E2 8842.344} C_VEL
LIN {X 0,Y 577.969,Z 767.06,A -85,B 0,C 180,E1 8851.487,E2 8851.487} C_VEL
LIN {X 0,Y 577.892,Z 768.512,A -85,B 0,C 180,E1 8858.511,E2 8858.511} C_VEL
LIN {X 0,Y 615.856,Z 830.61,A -85,B 0,C 180,E1 8863.949,E2 8863.949} C_VEL
LIN {X 0,Y 621.873,Z 844.951,A -85,B 0,C 180,E1 8864.847,E2 8864.847} C_VEL
LIN {X 0,Y 615.175,Z 921.093,A -85,B 0,C 180,E1 8867.026,E2 8867.026} C_VEL
LIN {X 0,Y 612.707,Z 944.277,A -85,B 0,C 180,E1 8868.027,E2 8868.027} C_VEL
LIN {X 0,Y 602.317,Z 976.103,A -85,B 0,C 180,E1 8869.145,E2 8869.145} C_VEL
LIN {X 0,Y 591.808,Z 1044.155,A -85,B 0,C 180,E1 8873.943,E2 8873.943} C_VEL
LIN {X 0,Y 582.267,Z 1103.279,A -85,B 0,C 180,E1 8880.079,E2 8880.079} C_VEL
LIN {X 0,Y 575.701,Z 1150.853,A -85,B 0,C 180,E1 8887.258,E2 8887.258} C_VEL
LIN {X 0,Y 572.575,Z 1185.315,A -85,B 0,C 180,E1 8895.17,E2 8895.17} C_VEL
LIN {X 0,Y 571.326,Z 1203.507,A -85,B 0,C 180,E1 8902.371,E2 8902.371} C_VEL
LIN {X 0,Y 570.765,Z 1209.837,A -85,B 0,C 180,E1 8909.237,E2 8909.237} C_VEL
LIN {X 0,Y 570.959,Z 1205.886,A -85,B 0,C 180,E1 8916.096,E2 8916.096} C_VEL
LIN {X 0,Y 571.57,Z 1191.034,A -85,B 0,C 180,E1 8923.031,E2 8923.031} C_VEL
LIN {X 0,Y 574.22,Z 1163.028,A -85,B 0,C 180,E1 8930.364,E2 8930.364} C_VEL
LIN {X 0,Y 579.861,Z 1120.319,A -85,B 0,C 180,E1 8937.656,E2 8937.656} C_VEL
LIN {X 0,Y 588.449,Z 1065.276,A -85,B 0,C 180,E1 8944.12,E2 8944.12} C_VEL
LIN {X 0,Y 598.714,Z 1000.505,A -85,B 0,C 180,E1 8949.359,E2 8949.359} C_VEL
LIN {X 0,Y 608.566,Z 928.65,A -85,B 0,C 180,E1 8953.171,E2 8953.171} C_VEL
LIN {X 0,Y 615.189,Z 859.753,A -85,B 0,C 180,E1 8955.374,E2 8955.374} C_VEL
LIN {X 0,Y 614.821,Z 841.717,A -85,B 0,C 180,E1 8955.897,E2 8955.897} C_VEL
LIN {X 0,Y 570.299,Z 767.06,A -85,B 0,C 180,E1 8962.304,E2 8962.304} C_VEL
LIN {X 0,Y 570.24,Z 767.06,A -85,B 0,C 180,E1 8970.538,E2 8970.538} C_VEL
LIN {X 0,Y 570.318,Z 767.06,A -85,B 0,C 180,E1 8980.598,E2 8980.598} C_VEL
LIN {X 0,Y 570.671,Z 767.06,A -85,B 0,C 180,E1 8990.066,E2 8990.066} C_VEL
LIN {X 0,Y 571.155,Z 767.06,A -85,B 0,C 180,E1 8997.732,E2 8997.732} C_VEL
LIN {X 0,Y 570.584,Z 767.06,A -85,B 0,C 180,E1 9006.886,E2 9006.886} C_VEL
LIN {X 0,Y 570.338,Z 767.06,A -85,B 0,C 180,E1 9014.651,E2 9014.651} C_VEL
LIN {X 0,Y 569.912,Z 767.06,A -85,B 0,C 180,E1 9023.371,E2 9023.371} C_VEL
LIN {X 0,Y 569.899,Z 767.06,A -85,B 0,C 180,E1 9031.284,E2 9031.284} C_VEL
LIN {X 0,Y 569.74,Z 767.06,A -85,B 0,C 180,E1 9040.734,E2 9040.734} C_VEL
LIN {X 0,Y 570.079,Z 768.152,A -85,B 0,C 180,E1 9043.942,E2 9043.942} C_VEL
LIN {X 0,Y 614.102,Z 841.665,A -85,B 0,C 180,E1 9050.23,E2 9050.23} C_VEL
LIN {X 0,Y 613.171,Z 873.413,A -85,B 0,C 180,E1 9051.172,E2 9051.172} C_VEL
LIN {X 0,Y 605.124,Z 946.085,A -85,B 0,C 180,E1 9054.024,E2 9054.024} C_VEL
LIN {X 0,Y 594.842,Z 1015.635,A -85,B 0,C 180,E1 9058.39,E2 9058.39} C_VEL
LIN {X 0,Y 584.713,Z 1077.433,A -85,B 0,C 180,E1 9064.147,E2 9064.147} C_VEL
LIN {X 0,Y 577.236,Z 1127.148,A -85,B 0,C 180,E1 9070.831,E2 9070.831} C_VEL
LIN {X 0,Y 573.11,Z 1164.332,A -85,B 0,C 180,E1 9078.149,E2 9078.149} C_VEL
LIN {X 0,Y 571.775,Z 1189.4,A -85,B 0,C 180,E1 9086.2,E2 9086.2} C_VEL
LIN {X 0,Y 570.972,Z 1199.481,A -85,B 0,C 180,E1 9093.809,E2 9093.809} C_VEL
LIN {X 0,Y 570.978,Z 1196.561,A -85,B 0,C 180,E1 9101.492,E2 9101.492} C_VEL
LIN {X 0,Y 571.971,Z 1181.097,A -85,B 0,C 180,E1 9108.955,E2 9108.955} C_VEL
LIN {X 0,Y 574.842,Z 1150.025,A -85,B 0,C 180,E1 9116.919,E2 9116.919} C_VEL
LIN {X 0,Y 580.471,Z 1106.218,A -85,B 0,C 180,E1 9124.175,E2 9124.175} C_VEL
LIN {X 0,Y 589.205,Z 1050.224,A -85,B 0,C 180,E1 9130.561,E2 9130.561} C_VEL
LIN {X 0,Y 599.598,Z 983.619,A -85,B 0,C 180,E1 9135.771,E2 9135.771} C_VEL
LIN {X 0,Y 609.407,Z 909.752,A -85,B 0,C 180,E1 9139.517,E2 9139.517} C_VEL
LIN {X 0,Y 614.396,Z 842.872,A -85,B 0,C 180,E1 9141.621,E2 9141.621} C_VEL
LIN {X 0,Y 580.279,Z 784.159,A -85,B 0,C 180,E1 9146.662,E2 9146.662} C_VEL
LIN {X 0,Y 570.146,Z 767.06,A -85,B 0,C 180,E1 9148.548,E2 9148.548} C_VEL
LIN {X 0,Y 570.327,Z 767.06,A -85,B 0,C 180,E1 9157.3,E2 9157.3} C_VEL
LIN {X 0,Y 571.086,Z 767.06,A -85,B 0,C 180,E1 9166.936,E2 9166.936} C_VEL
LIN {X 0,Y 571.21,Z 767.06,A -85,B 0,C 180,E1 9177.702,E2 9177.702} C_VEL
LIN {X 0,Y 570.522,Z 767.06,A -85,B 0,C 180,E1 9186.856,E2 9186.856} C_VEL
LIN {X 0,Y 570.36,Z 767.06,A -85,B 0,C 180,E1 9194.619,E2 9194.619} C_VEL
LIN {X 0,Y 569.988,Z 767.06,A -85,B 0,C 180,E1 9203.377,E2 9203.377} C_VEL
LIN {X 0,Y 570.002,Z 767.06,A -85,B 0,C 180,E1 9211.242,E2 9211.242} C_VEL
LIN {X 0,Y 569.89,Z 768.339,A -85,B 0,C 180,E1 9217.419,E2 9217.419} C_VEL
LIN {X 0,Y 609.158,Z 831.862,A -85,B 0,C 180,E1 9223.321,E2 9223.321} C_VEL
LIN {X 0,Y 616.019,Z 848.616,A -85,B 0,C 180,E1 9224.395,E2 9224.395} C_VEL
LIN {X 0,Y 608.916,Z 923.92,A -85,B 0,C 180,E1 9226.624,E2 9226.624} C_VEL
LIN {X 0,Y 602.317,Z 976.103,A -85,B 0,C 180,E1 9229.145,E2 9229.145} C_VEL
LIN {X 0,Y 591.388,Z 1006.551,A -85,B 0,C 180,E1 9230.538,E2 9230.538} C_VEL
LIN {X 0,Y 580.607,Z 1070.786,A -85,B 0,C 180,E1 9235.966,E2 9235.966} C_VEL
LIN {X 0,Y 571.581,Z 1125.552,A -85,B 0,C 180,E1 9242.717,E2 9242.717} C_VEL
LIN {X 0,Y 565.953,Z 1166.838,A -85,B 0,C 180,E1 9250.176,E2 9250.176} C_VEL
LIN {X 0,Y 563.421,Z 1193.288,A -85,B 0,C 180,E1 9257.563,E2 9257.563} C_VEL
LIN {X 0,Y 562.981,Z 1206.783,A -85,B 0,C 180,E1 9264.588,E2 9264.588} C_VEL
LIN {X 0,Y 562.644,Z 1209.838,A -85,B 0,C 180,E1 9270.77,E2 9270.77} C_VEL
LIN {X 0,Y 563.258,Z 1203.511,A -85,B 0,C 180,E1 9277.734,E2 9277.734} C_VEL
LIN {X 0,Y 564.743,Z 1183.525,A -85,B 0,C 180,E1 9285.574,E2 9285.574} C_VEL
LIN {X 0,Y 568.196,Z 1149.104,A -85,B 0,C 180,E1 9293.393,E2 9293.393} C_VEL
LIN {X 0,Y 575.171,Z 1102.048,A -85,B 0,C 180,E1 9300.497,E2 9300.497} C_VEL
LIN {X 0,Y 585.523,Z 1042.056,A -85,B 0,C 180,E1 9306.716,E2 9306.716} C_VEL
LIN {X 0,Y 596.185,Z 975.185,A -85,B 0,C 180,E1 9311.423,E2 9311.423} C_VEL
LIN {X 0,Y 605.508,Z 899.895,A -85,B 0,C 180,E1 9314.813,E2 9314.813} C_VEL
LIN {X 0,Y 609.119,Z 845.376,A -85,B 0,C 180,E1 9316.353,E2 9316.353} C_VEL
LIN {X 0,Y 564.01,Z 771.963,A -85,B 0,C 180,E1 9322.838,E2 9322.838} C_VEL
LIN {X 0,Y 562.313,Z 767.06,A -85,B 0,C 180,E1 9323.369,E2 9323.369} C_VEL
LIN {X 0,Y 562.202,Z 767.06,A -85,B 0,C 180,E1 9331.843,E2 9331.843} C_VEL
LIN {X 0,Y 562.333,Z 767.06,A -85,B 0,C 180,E1 9341.945,E2 9341.945} C_VEL
LIN {X 0,Y 562.461,Z 767.06,A -85,B 0,C 180,E1 9351.486,E2 9351.486} C_VEL
LIN {X 0,Y 562.587,Z 767.06,A -85,B 0,C 180,E1 9359.243,E2 9359.243} C_VEL
LIN {X 0,Y 562.554,Z 767.06,A -85,B 0,C 180,E1 9366.985,E2 9366.985} C_VEL
LIN {X 0,Y 562.283,Z 767.06,A -85,B 0,C 180,E1 9374.865,E2 9374.865} C_VEL
LIN {X 0,Y 561.942,Z 767.06,A -85,B 0,C 180,E1 9383.058,E2 9383.058} C_VEL
LIN {X 0,Y 561.824,Z 767.06,A -85,B 0,C 180,E1 9391.786,E2 9391.786} C_VEL
LIN {X 0,Y 561.698,Z 767.06,A -85,B 0,C 180,E1 9399.7,E2 9399.7} C_VEL
LIN {X 0,Y 562.124,Z 769.067,A -85,B 0,C 180,E1 9402.972,E2 9402.972} C_VEL
LIN {X 0,Y 605.899,Z 840.134,A -85,B 0,C 180,E1 9409.387,E2 9409.387} C_VEL
LIN {X 0,Y 609.411,Z 851.687,A -85,B 0,C 180,E1 9410.071,E2 9410.071} C_VEL
LIN {X 0,Y 602.177,Z 923.381,A -85,B 0,C 180,E1 9412.439,E2 9412.439} C_VEL
LIN {X 0,Y 591.954,Z 992.997,A -85,B 0,C 180,E1 9416.252,E2 9416.252} C_VEL
LIN {X 0,Y 580.9,Z 1058.287,A -85,B 0,C 180,E1 9421.657,E2 9421.657} C_VEL
LIN {X 0,Y 571.664,Z 1113.888,A -85,B 0,C 180,E1 9428.409,E2 9428.409} C_VEL
LIN {X 0,Y 566.012,Z 1154.766,A -85,B 0,C 180,E1 9435.653,E2 9435.653} C_VEL
LIN {X 0,Y 563.675,Z 1179.68,A -85,B 0,C 180,E1 9442.272,E2 9442.272} C_VEL
LIN {X 0,Y 562.961,Z 1193.889,A -85,B 0,C 180,E1 9448.459,E2 9448.459} C_VEL
LIN {X 0,Y 562.961,Z 1199.527,A -85,B 0,C 180,E1 9453.864,E2 9453.864} C_VEL
LIN {X 0,Y 563.001,Z 1196.462,A -85,B 0,C 180,E1 9461.657,E2 9461.657} C_VEL
LIN {X 0,Y 564.133,Z 1180.834,A -85,B 0,C 180,E1 9469.228,E2 9469.228} C_VEL
LIN {X 0,Y 567.049,Z 1149.846,A -85,B 0,C 180,E1 9477.258,E2 9477.258} C_VEL
LIN {X 0,Y 573.159,Z 1105.509,A -85,B 0,C 180,E1 9484.672,E2 9484.672} C_VEL
LIN {X 0,Y 582.561,Z 1049.289,A -85,B 0,C 180,E1 9491.115,E2 9491.115} C_VEL
LIN {X 0,Y 593.347,Z 983.385,A -85,B 0,C 180,E1 9496.298,E2 9496.298} C_VEL
LIN {X 0,Y 603.469,Z 910.138,A -85,B 0,C 180,E1 9500.038,E2 9500.038} C_VEL
LIN {X 0,Y 608.784,Z 846.69,A -85,B 0,C 180,E1 9502.062,E2 9502.062} C_VEL
LIN {X 0,Y 575.88,Z 789.148,A -85,B 0,C 180,E1 9507.133,E2 9507.133} C_VEL
LIN {X 0,Y 562.14,Z 767.06,A -85,B 0,C 180,E1 9509.693,E2 9509.693} C_VEL
LIN {X 0,Y 562.258,Z 767.06,A -85,B 0,C 180,E1 9518.625,E2 9518.625} C_VEL
LIN {X 0,Y 563.172,Z 767.06,A -85,B 0,C 180,E1 9528.33,E2 9528.33} C_VEL
LIN {X 0,Y 563.201,Z 767.06,A -85,B 0,C 180,E1 9537.669,E2 9537.669} C_VEL
LIN {X 0,Y 562.49,Z 767.06,A -85,B 0,C 180,E1 9546.954,E2 9546.954} C_VEL
LIN {X 0,Y 562.3,Z 767.06,A -85,B 0,C 180,E1 9554.833,E2 9554.833} C_VEL
LIN {X 0,Y 562.054,Z 767.06,A -85,B 0,C 180,E1 9563.02,E2 9563.02} C_VEL
LIN {X 0,Y 561.907,Z 767.06,A -85,B 0,C 180,E1 9571.772,E2 9571.772} C_VEL
LIN {X 0,Y 562.045,Z 769.071,A -85,B 0,C 180,E1 9576.302,E2 9576.302} C_VEL
LIN {X 0,Y 599.297,Z 827.663,A -85,B 0,C 180,E1 9582.226,E2 9582.226} C_VEL
LIN {X 0,Y 610.137,Z 853.037,A -85,B 0,C 180,E1 9583.947,E2 9583.947} C_VEL
LIN {X 0,Y 602.654,Z 926.746,A -85,B 0,C 180,E1 9586.21,E2 9586.21} C_VEL
LIN {X 0,Y 592.397,Z 999.461,A -85,B 0,C 180,E1 9590.061,E2 9590.061} C_VEL
LIN {X 0,Y 591.388,Z 1006.551,A -85,B 0,C 180,E1 9590.538,E2 9590.538} C_VEL
LIN {X 0,Y 579.966,Z 1035.433,A -85,B 0,C 180,E1 9592.222,E2 9592.222} C_VEL
LIN {X 0,Y 568.806,Z 1096.689,A -85,B 0,C 180,E1 9598.385,E2 9598.385} C_VEL
LIN {X 0,Y 560.95,Z 1144.694,A -85,B 0,C 180,E1 9605.438,E2 9605.438} C_VEL
LIN {X 0,Y 556.814,Z 1179.72,A -85,B 0,C 180,E1 9613.089,E2 9613.089} C_VEL
LIN {X 0,Y 555.517,Z 1200.603,A -85,B 0,C 180,E1 9620.571,E2 9620.571} C_VEL
LIN {X 0,Y 555.285,Z 1209.403,A -85,B 0,C 180,E1 9627.65,E2 9627.65} C_VEL
LIN {X 0,Y 555.049,Z 1206.786,A -85,B 0,C 180,E1 9635.485,E2 9635.485} C_VEL
LIN {X 0,Y 555.543,Z 1193.301,A -85,B 0,C 180,E1 9642.611,E2 9642.611} C_VEL
LIN {X 0,Y 558.149,Z 1166.628,A -85,B 0,C 180,E1 9650.162,E2 9650.162} C_VEL
LIN {X 0,Y 564.197,Z 1124.941,A -85,B 0,C 180,E1 9657.77,E2 9657.77} C_VEL
LIN {X 0,Y 573.516,Z 1071.489,A -85,B 0,C 180,E1 9664.43,E2 9664.43} C_VEL
LIN {X 0,Y 584.738,Z 1008.059,A -85,B 0,C 180,E1 9669.861,E2 9669.861} C_VEL
LIN {X 0,Y 595.698,Z 936.496,A -85,B 0,C 180,E1 9673.899,E2 9673.899} C_VEL
LIN {X 0,Y 603.341,Z 866.933,A -85,B 0,C 180,E1 9676.281,E2 9676.281} C_VEL
LIN {X 0,Y 603.339,Z 848.723,A -85,B 0,C 180,E1 9676.839,E2 9676.839} C_VEL
LIN {X 0,Y 557.309,Z 773.288,A -85,B 0,C 180,E1 9683.667,E2 9683.667} C_VEL
LIN {X 0,Y 554.284,Z 767.06,A -85,B 0,C 180,E1 9684.374,E2 9684.374} C_VEL
LIN {X 0,Y 554.128,Z 767.06,A -85,B 0,C 180,E1 9693.167,E2 9693.167} C_VEL
LIN {X 0,Y 554.287,Z 767.06,A -85,B 0,C 180,E1 9701.673,E2 9701.673} C_VEL
LIN {X 0,Y 554.482,Z 767.06,A -85,B 0,C 180,E1 9711.362,E2 9711.362} C_VEL
LIN {X 0,Y 554.589,Z 767.06,A -85,B 0,C 180,E1 9719.232,E2 9719.232} C_VEL
LIN {X 0,Y 554.548,Z 767.06,A -85,B 0,C 180,E1 9727.086,E2 9727.086} C_VEL
LIN {X 0,Y 554.247,Z 767.06,A -85,B 0,C 180,E1 9735.086,E2 9735.086} C_VEL
LIN {X 0,Y 553.869,Z 767.06,A -85,B 0,C 180,E1 9743.484,E2 9743.484} C_VEL
LIN {X 0,Y 553.747,Z 767.06,A -85,B 0,C 180,E1 9752.305,E2 9752.305} C_VEL
LIN {X 0,Y 553.864,Z 768.483,A -85,B 0,C 180,E1 9761.886,E2 9761.886} C_VEL
LIN {X 0,Y 598.606,Z 840.493,A -85,B 0,C 180,E1 9768.654,E2 9768.654} C_VEL
LIN {X 0,Y 603.614,Z 854.609,A -85,B 0,C 180,E1 9769.597,E2 9769.597} C_VEL
LIN {X 0,Y 596.039,Z 925.328,A -85,B 0,C 180,E1 9771.984,E2 9771.984} C_VEL
LIN {X 0,Y 585.44,Z 994.37,A -85,B 0,C 180,E1 9775.824,E2 9775.824} C_VEL
LIN {X 0,Y 573.679,Z 1060.159,A -85,B 0,C 180,E1 9781.375,E2 9781.375} C_VEL
LIN {X 0,Y 564.141,Z 1114.509,A -85,B 0,C 180,E1 9788.11,E2 9788.11} C_VEL
LIN {X 0,Y 558.193,Z 1155.158,A -85,B 0,C 180,E1 9795.448,E2 9795.448} C_VEL
LIN {X 0,Y 555.619,Z 1181.056,A -85,B 0,C 180,E1 9802.553,E2 9802.553} C_VEL
LIN {X 0,Y 554.783,Z 1195.221,A -85,B 0,C 180,E1 9809.219,E2 9809.219} C_VEL
LIN {X 0,Y 554.812,Z 1199.907,A -85,B 0,C 180,E1 9815.492,E2 9815.492} C_VEL
LIN {X 0,Y 555.349,Z 1194.086,A -85,B 0,C 180,E1 9823.423,E2 9823.423} C_VEL
LIN {X 0,Y 556.565,Z 1175.501,A -85,B 0,C 180,E1 9831.165,E2 9831.165} C_VEL
LIN {X 0,Y 559.755,Z 1142.99,A -85,B 0,C 180,E1 9838.967,E2 9838.967} C_VEL
LIN {X 0,Y 567.043,Z 1097.311,A -85,B 0,C 180,E1 9846.205,E2 9846.205} C_VEL
LIN {X 0,Y 577.506,Z 1038.836,A -85,B 0,C 180,E1 9852.573,E2 9852.573} C_VEL
LIN {X 0,Y 589.019,Z 972.673,A -85,B 0,C 180,E1 9857.473,E2 9857.473} C_VEL
LIN {X 0,Y 599.094,Z 898.317,A -85,B 0,C 180,E1 9861.023,E2 9861.023} C_VEL
LIN {X 0,Y 602.729,Z 849.701,A -85,B 0,C 180,E1 9862.565,E2 9862.565} C_VEL
LIN {X 0,Y 571.012,Z 793.172,A -85,B 0,C 180,E1 9867.702,E2 9867.702} C_VEL
LIN {X 0,Y 554.07,Z 767.06,A -85,B 0,C 180,E1 9870.813,E2 9870.813} C_VEL
LIN {X 0,Y 554.222,Z 767.06,A -85,B 0,C 180,E1 9879.978,E2 9879.978} C_VEL
LIN {X 0,Y 555.14,Z 767.06,A -85,B 0,C 180,E1 9888.159,E2 9888.159} C_VEL
LIN {X 0,Y 555.191,Z 767.06,A -85,B 0,C 180,E1 9897.636,E2 9897.636} C_VEL
LIN {X 0,Y 554.488,Z 767.06,A -85,B 0,C 180,E1 9907.055,E2 9907.055} C_VEL
LIN {X 0,Y 554.255,Z 767.06,A -85,B 0,C 180,E1 9915.053,E2 9915.053} C_VEL
LIN {X 0,Y 553.964,Z 767.06,A -85,B 0,C 180,E1 9923.496,E2 9923.496} C_VEL
LIN {X 0,Y 553.847,Z 767.06,A -85,B 0,C 180,E1 9932.262,E2 9932.262} C_VEL
LIN {X 0,Y 554.031,Z 769.041,A -85,B 0,C 180,E1 9935.07,E2 9935.07} C_VEL
LIN {X 0,Y 591.062,Z 826.072,A -85,B 0,C 180,E1 9941.282,E2 9941.282} C_VEL
LIN {X 0,Y 604.468,Z 855.114,A -85,B 0,C 180,E1 9943.447,E2 9943.447} C_VEL
LIN {X 0,Y 596.558,Z 928.504,A -85,B 0,C 180,E1 9945.744,E2 9945.744} C_VEL
LIN {X 0,Y 585.831,Z 1000.822,A -85,B 0,C 180,E1 9949.638,E2 9949.638} C_VEL
LIN {X 0,Y 579.966,Z 1035.433,A -85,B 0,C 180,E1 9952.222,E2 9952.222} C_VEL
LIN {X 0,Y 568.384,Z 1062.564,A -85,B 0,C 180,E1 9954.196,E2 9954.196} C_VEL
LIN {X 0,Y 558.074,Z 1118.435,A -85,B 0,C 180,E1 9960.88,E2 9960.88} C_VEL
LIN {X 0,Y 551.424,Z 1161.677,A -85,B 0,C 180,E1 9968.462,E2 9968.462} C_VEL
LIN {X 0,Y 547.913,Z 1191.01,A -85,B 0,C 180,E1 9976.391,E2 9976.391} C_VEL
LIN {X 0,Y 547.06,Z 1205.879,A -85,B 0,C 180,E1 9983.632,E2 9983.632} C_VEL
LIN {X 0,Y 546.777,Z 1209.837,A -85,B 0,C 180,E1 9989.203,E2 9989.203} C_VEL
LIN {X 0,Y 547.019,Z 1205.886,A -85,B 0,C 180,E1 9996.364,E2 9996.364} C_VEL
LIN {X 0,Y 548.098,Z 1189.494,A -85,B 0,C 180,E1 10004.143,E2 10004.143} C_VEL
LIN {X 0,Y 551.927,Z 1157.413,A -85,B 0,C 180,E1 10012.444,E2 10012.444} C_VEL
LIN {X 0,Y 559.278,Z 1111.546,A -85,B 0,C 180,E1 10020.105,E2 10020.105} C_VEL
LIN {X 0,Y 569.856,Z 1054.852,A -85,B 0,C 180,E1 10026.562,E2 10026.562} C_VEL
LIN {X 0,Y 581.75,Z 987.827,A -85,B 0,C 180,E1 10031.742,E2 10031.742} C_VEL
LIN {X 0,Y 592.747,Z 913.218,A -85,B 0,C 180,E1 10035.418,E2 10035.418} C_VEL
LIN {X 0,Y 597.543,Z 851.98,A -85,B 0,C 180,E1 10037.342,E2 10037.342} C_VEL
LIN {X 0,Y 553.343,Z 779.442,A -85,B 0,C 180,E1 10044.062,E2 10044.062} C_VEL
LIN {X 0,Y 546.25,Z 767.06,A -85,B 0,C 180,E1 10045.321,E2 10045.321} C_VEL
LIN {X 0,Y 546.022,Z 767.06,A -85,B 0,C 180,E1 10054.512,E2 10054.512} C_VEL
LIN {X 0,Y 546.282,Z 767.06,A -85,B 0,C 180,E1 10063.269,E2 10063.269} C_VEL
LIN {X 0,Y 546.48,Z 767.06,A -85,B 0,C 180,E1 10071.235,E2 10071.235} C_VEL
LIN {X 0,Y 546.603,Z 767.06,A -85,B 0,C 180,E1 10079.221,E2 10079.221} C_VEL
LIN {X 0,Y 546.521,Z 767.06,A -85,B 0,C 180,E1 10087.191,E2 10087.191} C_VEL
LIN {X 0,Y 546.201,Z 767.06,A -85,B 0,C 180,E1 10095.314,E2 10095.314} C_VEL
LIN {X 0,Y 545.848,Z 767.06,A -85,B 0,C 180,E1 10103.78,E2 10103.78} C_VEL
LIN {X 0,Y 545.733,Z 767.06,A -85,B 0,C 180,E1 10112.839,E2 10112.839} C_VEL
LIN {X 0,Y 545.834,Z 768.778,A -85,B 0,C 180,E1 10120.794,E2 10120.794} C_VEL
LIN {X 0,Y 589.404,Z 837.676,A -85,B 0,C 180,E1 10127.607,E2 10127.607} C_VEL
LIN {X 0,Y 597.858,Z 857.382,A -85,B 0,C 180,E1 10129.108,E2 10129.108} C_VEL
LIN {X 0,Y 589.763,Z 928.223,A -85,B 0,C 180,E1 10131.564,E2 10131.564} C_VEL
LIN {X 0,Y 578.672,Z 997.099,A -85,B 0,C 180,E1 10135.482,E2 10135.482} C_VEL
LIN {X 0,Y 566.654,Z 1061.001,A -85,B 0,C 180,E1 10140.987,E2 10140.987} C_VEL
LIN {X 0,Y 556.647,Z 1115.1,A -85,B 0,C 180,E1 10147.8,E2 10147.8} C_VEL
LIN {X 0,Y 550.368,Z 1155.55,A -85,B 0,C 180,E1 10155.236,E2 10155.236} C_VEL
LIN {X 0,Y 547.664,Z 1181.305,A -85,B 0,C 180,E1 10162.445,E2 10162.445} C_VEL
LIN {X 0,Y 546.803,Z 1195.35,A -85,B 0,C 180,E1 10169.208,E2 10169.208} C_VEL
LIN {X 0,Y 546.805,Z 1199.926,A -85,B 0,C 180,E1 10175.573,E2 10175.573} C_VEL
LIN {X 0,Y 547.254,Z 1195.177,A -85,B 0,C 180,E1 10182.81,E2 10182.81} C_VEL
LIN {X 0,Y 548.613,Z 1176.57,A -85,B 0,C 180,E1 10191.062,E2 10191.062} C_VEL
LIN {X 0,Y 551.945,Z 1144.062,A -85,B 0,C 180,E1 10199.099,E2 10199.099} C_VEL
LIN {X 0,Y 559.613,Z 1098.439,A -85,B 0,C 180,E1 10206.49,E2 10206.49} C_VEL
LIN {X 0,Y 570.708,Z 1039.499,A -85,B 0,C 180,E1 10213.015,E2 10213.015} C_VEL
LIN {X 0,Y 582.894,Z 972.749,A -85,B 0,C 180,E1 10218.008,E2 10218.008} C_VEL
LIN {X 0,Y 593.388,Z 898.423,A -85,B 0,C 180,E1 10221.575,E2 10221.575} C_VEL
LIN {X 0,Y 596.971,Z 853.284,A -85,B 0,C 180,E1 10223.034,E2 10223.034} C_VEL
LIN {X 0,Y 567.247,Z 799.238,A -85,B 0,C 180,E1 10228.093,E2 10228.093} C_VEL
LIN {X 0,Y 545.998,Z 767.06,A -85,B 0,C 180,E1 10232.393,E2 10232.393} C_VEL
LIN {X 0,Y 546.232,Z 767.06,A -85,B 0,C 180,E1 10241.36,E2 10241.36} C_VEL
LIN {X 0,Y 546.931,Z 767.06,A -85,B 0,C 180,E1 10249.845,E2 10249.845} C_VEL
LIN {X 0,Y 546.638,Z 767.06,A -85,B 0,C 180,E1 10259.189,E2 10259.189} C_VEL
LIN {X 0,Y 546.457,Z 767.06,A -85,B 0,C 180,E1 10267.16,E2 10267.16} C_VEL
LIN {X 0,Y 546.204,Z 767.06,A -85,B 0,C 180,E1 10275.281,E2 10275.281} C_VEL
LIN {X 0,Y 545.94,Z 767.06,A -85,B 0,C 180,E1 10283.74,E2 10283.74} C_VEL
LIN {X 0,Y 545.822,Z 767.06,A -85,B 0,C 180,E1 10292.795,E2 10292.795} C_VEL
LIN {X 0,Y 546.045,Z 769.109,A -85,B 0,C 180,E1 10293.759,E2 10293.759} C_VEL
LIN {X 0,Y 580.99,Z 821.787,A -85,B 0,C 180,E1 10299.99,E2 10299.99} C_VEL
LIN {X 0,Y 598.576,Z 858.855,A -85,B 0,C 180,E1 10302.977,E2 10302.977} C_VEL
LIN {X 0,Y 590.289,Z 932.643,A -85,B 0,C 180,E1 10305.375,E2 10305.375} C_VEL
LIN {X 0,Y 578.829,Z 1005.17,A -85,B 0,C 180,E1 10309.407,E2 10309.407} C_VEL
LIN {X 0,Y 568.384,Z 1062.564,A -85,B 0,C 180,E1 10314.196,E2 10314.196} C_VEL
LIN {X 0,Y 556.373,Z 1087.862,A -85,B 0,C 180,E1 10316.424,E2 10316.424} C_VEL
LIN {X 0,Y 546.901,Z 1138.67,A -85,B 0,C 180,E1 10323.66,E2 10323.66} C_VEL
LIN {X 0,Y 541.464,Z 1174.679,A -85,B 0,C 180,E1 10331.209,E2 10331.209} C_VEL
LIN {X 0,Y 539.403,Z 1195.277,A -85,B 0,C 180,E1 10337.825,E2 10337.825} C_VEL
LIN {X 0,Y 539.008,Z 1206.774,A -85,B 0,C 180,E1 10344.347,E2 10344.347} C_VEL
LIN {X 0,Y 538.662,Z 1209.838,A -85,B 0,C 180,E1 10350.804,E2 10350.804} C_VEL
LIN {X 0,Y 539.383,Z 1203.503,A -85,B 0,C 180,E1 10358.079,E2 10358.079} C_VEL
LIN {X 0,Y 540.954,Z 1183.523,A -85,B 0,C 180,E1 10366.277,E2 10366.277} C_VEL
LIN {X 0,Y 545.112,Z 1149.178,A -85,B 0,C 180,E1 10374.431,E2 10374.431} C_VEL
LIN {X 0,Y 553.456,Z 1102.446,A -85,B 0,C 180,E1 10381.772,E2 10381.772} C_VEL
LIN {X 0,Y 565.16,Z 1044.205,A -85,B 0,C 180,E1 10388.029,E2 10388.029} C_VEL
LIN {X 0,Y 577.714,Z 975.969,A -85,B 0,C 180,E1 10392.977,E2 10392.977} C_VEL
LIN {X 0,Y 588.368,Z 900.342,A -85,B 0,C 180,E1 10396.457,E2 10396.457} C_VEL
LIN {X 0,Y 591.946,Z 855.649,A -85,B 0,C 180,E1 10397.82,E2 10397.82} C_VEL
LIN {X 0,Y 549.392,Z 785.35,A -85,B 0,C 180,E1 10404.469,E2 10404.469} C_VEL
LIN {X 0,Y 538.148,Z 767.06,A -85,B 0,C 180,E1 10406.677,E2 10406.677} C_VEL
LIN {X 0,Y 537.952,Z 767.06,A -85,B 0,C 180,E1 10416.365,E2 10416.365} C_VEL
LIN {X 0,Y 538.175,Z 767.06,A -85,B 0,C 180,E1 10424.486,E2 10424.486} C_VEL
LIN {X 0,Y 538.308,Z 767.06,A -85,B 0,C 180,E1 10432.731,E2 10432.731} C_VEL
LIN {X 0,Y 538.626,Z 767.06,A -85,B 0,C 180,E1 10439.209,E2 10439.209} C_VEL
LIN {X 0,Y 538.495,Z 767.06,A -85,B 0,C 180,E1 10447.299,E2 10447.299} C_VEL
LIN {X 0,Y 538.176,Z 767.06,A -85,B 0,C 180,E1 10455.548,E2 10455.548} C_VEL
LIN {X 0,Y 537.821,Z 767.06,A -85,B 0,C 180,E1 10464.157,E2 10464.157} C_VEL
LIN {X 0,Y 537.641,Z 767.06,A -85,B 0,C 180,E1 10473.692,E2 10473.692} C_VEL
LIN {X 0,Y 537.796,Z 768.576,A -85,B 0,C 180,E1 10479.63,E2 10479.63} C_VEL
LIN {X 0,Y 580.975,Z 836.323,A -85,B 0,C 180,E1 10486.655,E2 10486.655} C_VEL
LIN {X 0,Y 592.09,Z 860.788,A -85,B 0,C 180,E1 10488.626,E2 10488.626} C_VEL
LIN {X 0,Y 583.581,Z 930.819,A -85,B 0,C 180,E1 10491.124,E2 10491.124} C_VEL
LIN {X 0,Y 571.898,Z 999.695,A -85,B 0,C 180,E1 10495.13,E2 10495.13} C_VEL
LIN {X 0,Y 559.205,Z 1063.91,A -85,B 0,C 180,E1 10500.813,E2 10500.813} C_VEL
LIN {X 0,Y 548.663,Z 1118.233,A -85,B 0,C 180,E1 10507.885,E2 10507.885} C_VEL
LIN {X 0,Y 542.321,Z 1157.691,A -85,B 0,C 180,E1 10515.439,E2 10515.439} C_VEL
LIN {X 0,Y 539.642,Z 1182.681,A -85,B 0,C 180,E1 10522.738,E2 10522.738} C_VEL
LIN {X 0,Y 538.806,Z 1195.477,A -85,B 0,C 180,E1 10529.196,E2 10529.196} C_VEL
LIN {X 0,Y 538.805,Z 1199.944,A -85,B 0,C 180,E1 10535.656,E2 10535.656} C_VEL
LIN {X 0,Y 539.375,Z 1193.809,A -85,B 0,C 180,E1 10543.829,E2 10543.829} C_VEL
LIN {X 0,Y 540.6,Z 1174.871,A -85,B 0,C 180,E1 10551.822,E2 10551.822} C_VEL
LIN {X 0,Y 544.316,Z 1143.673,A -85,B 0,C 180,E1 10559.521,E2 10559.521} C_VEL
LIN {X 0,Y 552.404,Z 1098.27,A -85,B 0,C 180,E1 10566.956,E2 10566.956} C_VEL
LIN {X 0,Y 563.969,Z 1040.146,A -85,B 0,C 180,E1 10573.474,E2 10573.474} C_VEL
LIN {X 0,Y 576.573,Z 974.306,A -85,B 0,C 180,E1 10578.465,E2 10578.465} C_VEL
LIN {X 0,Y 587.395,Z 901.534,A -85,B 0,C 180,E1 10582.03,E2 10582.03} C_VEL
LIN {X 0,Y 591.258,Z 856.768,A -85,B 0,C 180,E1 10583.524,E2 10583.524} C_VEL
LIN {X 0,Y 563.033,Z 804.59,A -85,B 0,C 180,E1 10588.573,E2 10588.573} C_VEL
LIN {X 0,Y 538,Z 767.06,A -85,B 0,C 180,E1 10593.619,E2 10593.619} C_VEL
LIN {X 0,Y 538.364,Z 767.06,A -85,B 0,C 180,E1 10602.775,E2 10602.775} C_VEL
LIN {X 0,Y 538.653,Z 767.06,A -85,B 0,C 180,E1 10611.074,E2 10611.074} C_VEL
LIN {X 0,Y 538.65,Z 767.06,A -85,B 0,C 180,E1 10619.177,E2 10619.177} C_VEL
LIN {X 0,Y 538.428,Z 767.06,A -85,B 0,C 180,E1 10627.267,E2 10627.267} C_VEL
LIN {X 0,Y 538.171,Z 767.06,A -85,B 0,C 180,E1 10635.514,E2 10635.514} C_VEL
LIN {X 0,Y 537.905,Z 767.06,A -85,B 0,C 180,E1 10644.117,E2 10644.117} C_VEL
LIN {X 0,Y 538.027,Z 768.83,A -85,B 0,C 180,E1 10652.337,E2 10652.337} C_VEL
LIN {X 0,Y 572.74,Z 820.623,A -85,B 0,C 180,E1 10658.913,E2 10658.913} C_VEL
LIN {X 0,Y 592.917,Z 861.112,A -85,B 0,C 180,E1 10662.46,E2 10662.46} C_VEL
LIN {X 0,Y 584.123,Z 935.074,A -85,B 0,C 180,E1 10664.93,E2 10664.93} C_VEL
LIN {X 0,Y 572.202,Z 1006.837,A -85,B 0,C 180,E1 10668.996,E2 10668.996} C_VEL
LIN {X 0,Y 559.767,Z 1071.581,A -85,B 0,C 180,E1 10674.612,E2 10674.612} C_VEL
LIN {X 0,Y 556.373,Z 1087.862,A -85,B 0,C 180,E1 10676.424,E2 10676.424} C_VEL
LIN {X 0,Y 544.741,Z 1111.118,A -85,B 0,C 180,E1 10678.938,E2 10678.938} C_VEL
LIN {X 0,Y 536.56,Z 1156.662,A -85,B 0,C 180,E1 10686.707,E2 10686.707} C_VEL
LIN {X 0,Y 532.583,Z 1188.966,A -85,B 0,C 180,E1 10695.245,E2 10695.245} C_VEL
LIN {X 0,Y 531.112,Z 1205.879,A -85,B 0,C 180,E1 10703.44,E2 10703.44} C_VEL
LIN {X 0,Y 530.797,Z 1209.836,A -85,B 0,C 180,E1 10709.179,E2 10709.179} C_VEL
LIN {X 0,Y 531.067,Z 1205.886,A -85,B 0,C 180,E1 10716.556,E2 10716.556} C_VEL
LIN {X 0,Y 532.396,Z 1189.188,A -85,B 0,C 180,E1 10724.68,E2 10724.68} C_VEL
LIN {X 0,Y 536.386,Z 1158.545,A -85,B 0,C 180,E1 10732.875,E2 10732.875} C_VEL
LIN {X 0,Y 544.258,Z 1114.058,A -85,B 0,C 180,E1 10740.626,E2 10740.626} C_VEL
LIN {X 0,Y 555.761,Z 1058.028,A -85,B 0,C 180,E1 10747.256,E2 10747.256} C_VEL
LIN {X 0,Y 568.718,Z 991.751,A -85,B 0,C 180,E1 10752.576,E2 10752.576} C_VEL
LIN {X 0,Y 580.775,Z 917.618,A -85,B 0,C 180,E1 10756.376,E2 10756.376} C_VEL
LIN {X 0,Y 586.035,Z 858.995,A -85,B 0,C 180,E1 10758.327,E2 10758.327} C_VEL
LIN {X 0,Y 545.27,Z 790.922,A -85,B 0,C 180,E1 10764.916,E2 10764.916} C_VEL
LIN {X 0,Y 530.085,Z 767.06,A -85,B 0,C 180,E1 10767.835,E2 10767.835} C_VEL
LIN {X 0,Y 529.925,Z 767.06,A -85,B 0,C 180,E1 10777.286,E2 10777.286} C_VEL
LIN {X 0,Y 530.181,Z 767.06,A -85,B 0,C 180,E1 10785.942,E2 10785.942} C_VEL
LIN {X 0,Y 530.892,Z 767.06,A -85,B 0,C 180,E1 10795.92,E2 10795.92} C_VEL
LIN {X 0,Y 530.854,Z 767.06,A -85,B 0,C 180,E1 10805.756,E2 10805.756} C_VEL
LIN {X 0,Y 530.132,Z 767.06,A -85,B 0,C 180,E1 10815.79,E2 10815.79} C_VEL
LIN {X 0,Y 529.769,Z 767.06,A -85,B 0,C 180,E1 10824.548,E2 10824.548} C_VEL
LIN {X 0,Y 529.643,Z 767.06,A -85,B 0,C 180,E1 10833.97,E2 10833.97} C_VEL
LIN {X 0,Y 529.774,Z 768.685,A -85,B 0,C 180,E1 10838.41,E2 10838.41} C_VEL
LIN {X 0,Y 571.465,Z 833.096,A -85,B 0,C 180,E1 10845.486,E2 10845.486} C_VEL
LIN {X 0,Y 586.379,Z 863.283,A -85,B 0,C 180,E1 10848.112,E2 10848.112} C_VEL
LIN {X 0,Y 577.327,Z 934.138,A -85,B 0,C 180,E1 10850.708,E2 10850.708} C_VEL
LIN {X 0,Y 564.957,Z 1003.334,A -85,B 0,C 180,E1 10854.848,E2 10854.848} C_VEL
LIN {X 0,Y 551.759,Z 1066.793,A -85,B 0,C 180,E1 10860.623,E2 10860.623} C_VEL
LIN {X 0,Y 540.931,Z 1120.067,A -85,B 0,C 180,E1 10867.764,E2 10867.764} C_VEL
LIN {X 0,Y 534.44,Z 1158.477,A -85,B 0,C 180,E1 10875.32,E2 10875.32} C_VEL
LIN {X 0,Y 531.673,Z 1182.927,A -85,B 0,C 180,E1 10882.628,E2 10882.628} C_VEL
LIN {X 0,Y 530.833,Z 1195.599,A -85,B 0,C 180,E1 10889.184,E2 10889.184} C_VEL
LIN {X 0,Y 530.798,Z 1199.963,A -85,B 0,C 180,E1 10895.741,E2 10895.741} C_VEL
LIN {X 0,Y 531.3,Z 1194.901,A -85,B 0,C 180,E1 10903.202,E2 10903.202} C_VEL
LIN {X 0,Y 532.66,Z 1176.553,A -85,B 0,C 180,E1 10911.531,E2 10911.531} C_VEL
LIN {X 0,Y 536.525,Z 1144.827,A -85,B 0,C 180,E1 10919.648,E2 10919.648} C_VEL
LIN {X 0,Y 544.894,Z 1100.105,A -85,B 0,C 180,E1 10927.163,E2 10927.163} C_VEL
LIN {X 0,Y 556.918,Z 1042.601,A -85,B 0,C 180,E1 10933.777,E2 10933.777} C_VEL
LIN {X 0,Y 570.021,Z 977.477,A -85,B 0,C 180,E1 10938.834,E2 10938.834} C_VEL
LIN {X 0,Y 581.594,Z 903.691,A -85,B 0,C 180,E1 10942.534,E2 10942.534} C_VEL
LIN {X 0,Y 585.627,Z 860.12,A -85,B 0,C 180,E1 10944.032,E2 10944.032} C_VEL
LIN {X 0,Y 558.418,Z 809.17,A -85,B 0,C 180,E1 10949.137,E2 10949.137} C_VEL
LIN {X 0,Y 530.035,Z 767.06,A -85,B 0,C 180,E1 10955.202,E2 10955.202} C_VEL
LIN {X 0,Y 530.556,Z 767.06,A -85,B 0,C 180,E1 10964.223,E2 10964.223} C_VEL
LIN {X 0,Y 530.399,Z 767.06,A -85,B 0,C 180,E1 10972.589,E2 10972.589} C_VEL
LIN {X 0,Y 530.672,Z 767.06,A -85,B 0,C 180,E1 10979.165,E2 10979.165} C_VEL
LIN {X 0,Y 530.401,Z 767.06,A -85,B 0,C 180,E1 10987.378,E2 10987.378} C_VEL
LIN {X 0,Y 530.044,Z 767.06,A -85,B 0,C 180,E1 10996.569,E2 10996.569} C_VEL
LIN {X 0,Y 529.823,Z 767.06,A -85,B 0,C 180,E1 11005.627,E2 11005.627} C_VEL
LIN {X 0,Y 530.085,Z 768.944,A -85,B 0,C 180,E1 11010.825,E2 11010.825} C_VEL
LIN {X 0,Y 564.142,Z 818.535,A -85,B 0,C 180,E1 11017.695,E2 11017.695} C_VEL
LIN {X 0,Y 587.362,Z 863.511,A -85,B 0,C 180,E1 11021.936,E2 11021.936} C_VEL
LIN {X 0,Y 578.116,Z 936.711,A -85,B 0,C 180,E1 11024.438,E2 11024.438} C_VEL
LIN {X 0,Y 565.524,Z 1008.911,A -85,B 0,C 180,E1 11028.605,E2 11028.605} C_VEL
LIN {X 0,Y 552.666,Z 1072.688,A -85,B 0,C 180,E1 11034.24,E2 11034.24} C_VEL
LIN {X 0,Y 544.741,Z 1111.118,A -85,B 0,C 180,E1 11038.938,E2 11038.938} C_VEL
LIN {X 0,Y 533.341,Z 1132.179,A -85,B 0,C 180,E1 11041.739,E2 11041.739} C_VEL
LIN {X 0,Y 526.318,Z 1172.173,A -85,B 0,C 180,E1 11049.968,E2 11049.968} C_VEL
LIN {X 0,Y 523.519,Z 1195.271,A -85,B 0,C 180,E1 11057.45,E2 11057.45} C_VEL
LIN {X 0,Y 523.018,Z 1206.768,A -85,B 0,C 180,E1 11064.173,E2 11064.173} C_VEL
LIN {X 0,Y 522.704,Z 1209.837,A -85,B 0,C 180,E1 11070.829,E2 11070.829} C_VEL
LIN {X 0,Y 523.424,Z 1203.497,A -85,B 0,C 180,E1 11078.327,E2 11078.327} C_VEL
LIN {X 0,Y 525.073,Z 1183.521,A -85,B 0,C 180,E1 11086.784,E2 11086.784} C_VEL
LIN {X 0,Y 529.585,Z 1150.858,A -85,B 0,C 180,E1 11094.846,E2 11094.846} C_VEL
LIN {X 0,Y 538.859,Z 1104.283,A -85,B 0,C 180,E1 11102.46,E2 11102.46} C_VEL
LIN {X 0,Y 551.94,Z 1044.605,A -85,B 0,C 180,E1 11109.044,E2 11109.044} C_VEL
LIN {X 0,Y 565.619,Z 976.695,A -85,B 0,C 180,E1 11114.056,E2 11114.056} C_VEL
LIN {X 0,Y 577.019,Z 901.752,A -85,B 0,C 180,E1 11117.557,E2 11117.557} C_VEL
LIN {X 0,Y 580.327,Z 862.798,A -85,B 0,C 180,E1 11118.805,E2 11118.805} C_VEL
LIN {X 0,Y 541.399,Z 796.769,A -85,B 0,C 180,E1 11125.332,E2 11125.332} C_VEL
LIN {X 0,Y 522.044,Z 767.06,A -85,B 0,C 180,E1 11129.208,E2 11129.208} C_VEL
LIN {X 0,Y 521.97,Z 767.06,A -85,B 0,C 180,E1 11138.718,E2 11138.718} C_VEL
LIN {X 0,Y 522.33,Z 767.06,A -85,B 0,C 180,E1 11147.437,E2 11147.437} C_VEL
LIN {X 0,Y 523.136,Z 767.06,A -85,B 0,C 180,E1 11157.524,E2 11157.524} C_VEL
LIN {X 0,Y 522.829,Z 767.06,A -85,B 0,C 180,E1 11165.845,E2 11165.845} C_VEL
LIN {X 0,Y 522.305,Z 767.06,A -85,B 0,C 180,E1 11174.309,E2 11174.309} C_VEL
LIN {X 0,Y 521.76,Z 767.06,A -85,B 0,C 180,E1 11183.726,E2 11183.726} C_VEL
LIN {X 0,Y 521.662,Z 767.06,A -85,B 0,C 180,E1 11192.563,E2 11192.563} C_VEL
LIN {X 0,Y 521.79,Z 768.978,A -85,B 0,C 180,E1 11197.125,E2 11197.125} C_VEL
LIN {X 0,Y 562.835,Z 831.233,A -85,B 0,C 180,E1 11204.408,E2 11204.408} C_VEL
LIN {X 0,Y 580.52,Z 867.452,A -85,B 0,C 180,E1 11207.64,E2 11207.64} C_VEL
LIN {X 0,Y 570.979,Z 938.268,A -85,B 0,C 180,E1 11210.324,E2 11210.324} C_VEL
LIN {X 0,Y 558.299,Z 1005.644,A -85,B 0,C 180,E1 11214.46,E2 11214.46} C_VEL
LIN {X 0,Y 544.627,Z 1068.453,A -85,B 0,C 180,E1 11220.293,E2 11220.293} C_VEL
LIN {X 0,Y 533.205,Z 1121.929,A -85,B 0,C 180,E1 11227.645,E2 11227.645} C_VEL
LIN {X 0,Y 526.374,Z 1160.716,A -85,B 0,C 180,E1 11235.558,E2 11235.558} C_VEL
LIN {X 0,Y 523.614,Z 1185.144,A -85,B 0,C 180,E1 11243.35,E2 11243.35} C_VEL
LIN {X 0,Y 523.149,Z 1197.495,A -85,B 0,C 180,E1 11250.833,E2 11250.833} C_VEL
LIN {X 0,Y 522.889,Z 1198.95,A -85,B 0,C 180,E1 11259.181,E2 11259.181} C_VEL
LIN {X 0,Y 523.428,Z 1188.434,A -85,B 0,C 180,E1 11267.107,E2 11267.107} C_VEL
LIN {X 0,Y 525.622,Z 1166.794,A -85,B 0,C 180,E1 11274.732,E2 11274.732} C_VEL
LIN {X 0,Y 531.644,Z 1130.288,A -85,B 0,C 180,E1 11282.803,E2 11282.803} C_VEL
LIN {X 0,Y 542.333,Z 1079.099,A -85,B 0,C 180,E1 11290.365,E2 11290.365} C_VEL
LIN {X 0,Y 555.592,Z 1018.356,A -85,B 0,C 180,E1 11296.456,E2 11296.456} C_VEL
LIN {X 0,Y 569.267,Z 948.709,A -85,B 0,C 180,E1 11301.062,E2 11301.062} C_VEL
LIN {X 0,Y 579.639,Z 878.707,A -85,B 0,C 180,E1 11303.954,E2 11303.954} C_VEL
LIN {X 0,Y 579.953,Z 863.463,A -85,B 0,C 180,E1 11304.567,E2 11304.567} C_VEL
LIN {X 0,Y 553.212,Z 812.526,A -85,B 0,C 180,E1 11309.832,E2 11309.832} C_VEL
LIN {X 0,Y 523.499,Z 771.623,A -85,B 0,C 180,E1 11316.247,E2 11316.247} C_VEL
LIN {X 0,Y 522.105,Z 767.06,A -85,B 0,C 180,E1 11316.89,E2 11316.89} C_VEL
LIN {X 0,Y 523.013,Z 767.06,A -85,B 0,C 180,E1 11327.42,E2 11327.42} C_VEL
LIN {X 0,Y 523.191,Z 767.06,A -85,B 0,C 180,E1 11337.491,E2 11337.491} C_VEL
LIN {X 0,Y 522.76,Z 767.06,A -85,B 0,C 180,E1 11345.812,E2 11345.812} C_VEL
LIN {X 0,Y 522.296,Z 767.06,A -85,B 0,C 180,E1 11354.274,E2 11354.274} C_VEL
LIN {X 0,Y 521.845,Z 767.06,A -85,B 0,C 180,E1 11363.735,E2 11363.735} C_VEL
LIN {X 0,Y 522.047,Z 768.761,A -85,B 0,C 180,E1 11369.152,E2 11369.152} C_VEL
LIN {X 0,Y 555.692,Z 816.96,A -85,B 0,C 180,E1 11376.43,E2 11376.43} C_VEL
LIN {X 0,Y 581.8,Z 866.131,A -85,B 0,C 180,E1 11381.398,E2 11381.398} C_VEL
LIN {X 0,Y 572.32,Z 937.513,A -85,B 0,C 180,E1 11383.889,E2 11383.889} C_VEL
LIN {X 0,Y 559.1,Z 1009.811,A -85,B 0,C 180,E1 11388.118,E2 11388.118} C_VEL
LIN {X 0,Y 545.737,Z 1073.153,A -85,B 0,C 180,E1 11393.788,E2 11393.788} C_VEL
LIN {X 0,Y 534.767,Z 1125.815,A -85,B 0,C 180,E1 11400.712,E2 11400.712} C_VEL
LIN {X 0,Y 533.341,Z 1132.179,A -85,B 0,C 180,E1 11401.739,E2 11401.739} C_VEL
LIN {X 0,Y 521.965,Z 1150.919,A -85,B 0,C 180,E1 11404.778,E2 11404.778} C_VEL
LIN {X 0,Y 517.055,Z 1183.923,A -85,B 0,C 180,E1 11413.081,E2 11413.081} C_VEL
LIN {X 0,Y 515.508,Z 1203.486,A -85,B 0,C 180,E1 11421.54,E2 11421.54} C_VEL
LIN {X 0,Y 514.799,Z 1209.836,A -85,B 0,C 180,E1 11429.154,E2 11429.154} C_VEL
LIN {X 0,Y 515.095,Z 1205.886,A -85,B 0,C 180,E1 11436.76,E2 11436.76} C_VEL
LIN {X 0,Y 516.728,Z 1188.714,A -85,B 0,C 180,E1 11445.312,E2 11445.312} C_VEL
LIN {X 0,Y 521.099,Z 1157.885,A -85,B 0,C 180,E1 11453.739,E2 11453.739} C_VEL
LIN {X 0,Y 529.927,Z 1113.241,A -85,B 0,C 180,E1 11461.67,E2 11461.67} C_VEL
LIN {X 0,Y 542.675,Z 1057.082,A -85,B 0,C 180,E1 11468.404,E2 11468.404} C_VEL
LIN {X 0,Y 556.661,Z 991.486,A -85,B 0,C 180,E1 11473.731,E2 11473.731} C_VEL
LIN {X 0,Y 569.511,Z 917.398,A -85,B 0,C 180,E1 11477.551,E2 11477.551} C_VEL
LIN {X 0,Y 574.634,Z 866.607,A -85,B 0,C 180,E1 11479.292,E2 11479.292} C_VEL
LIN {X 0,Y 537.923,Z 803.125,A -85,B 0,C 180,E1 11485.689,E2 11485.689} C_VEL
LIN {X 0,Y 513.988,Z 767.06,A -85,B 0,C 180,E1 11490.496,E2 11490.496} C_VEL
LIN {X 0,Y 514.061,Z 767.06,A -85,B 0,C 180,E1 11500.182,E2 11500.182} C_VEL
LIN {X 0,Y 514.48,Z 767.06,A -85,B 0,C 180,E1 11508.969,E2 11508.969} C_VEL
LIN {X 0,Y 515.121,Z 767.06,A -85,B 0,C 180,E1 11517.485,E2 11517.485} C_VEL
LIN {X 0,Y 514.793,Z 767.06,A -85,B 0,C 180,E1 11525.936,E2 11525.936} C_VEL
LIN {X 0,Y 514.249,Z 767.06,A -85,B 0,C 180,E1 11534.538,E2 11534.538} C_VEL
LIN {X 0,Y 513.776,Z 767.06,A -85,B 0,C 180,E1 11543.507,E2 11543.507} C_VEL
LIN {X 0,Y 513.636,Z 767.06,A -85,B 0,C 180,E1 11553.136,E2 11553.136} C_VEL
LIN {X 0,Y 513.756,Z 768.958,A -85,B 0,C 180,E1 11555.74,E2 11555.74} C_VEL
LIN {X 0,Y 554.184,Z 829.37,A -85,B 0,C 180,E1 11563.275,E2 11563.275} C_VEL
LIN {X 0,Y 574.735,Z 870.161,A -85,B 0,C 180,E1 11567.125,E2 11567.125} C_VEL
LIN {X 0,Y 564.715,Z 941.835,A -85,B 0,C 180,E1 11569.908,E2 11569.908} C_VEL
LIN {X 0,Y 551.473,Z 1008.996,A -85,B 0,C 180,E1 11574.143,E2 11574.143} C_VEL
LIN {X 0,Y 536.983,Z 1072.359,A -85,B 0,C 180,E1 11580.207,E2 11580.207} C_VEL
LIN {X 0,Y 525.487,Z 1123.668,A -85,B 0,C 180,E1 11587.5,E2 11587.5} C_VEL
LIN {X 0,Y 518.392,Z 1162.168,A -85,B 0,C 180,E1 11595.605,E2 11595.605} C_VEL
LIN {X 0,Y 515.655,Z 1185.352,A -85,B 0,C 180,E1 11603.247,E2 11603.247} C_VEL
LIN {X 0,Y 515.149,Z 1197.587,A -85,B 0,C 180,E1 11610.846,E2 11610.846} C_VEL
LIN {X 0,Y 514.906,Z 1198.973,A -85,B 0,C 180,E1 11619.189,E2 11619.189} C_VEL
LIN {X 0,Y 515.436,Z 1189.144,A -85,B 0,C 180,E1 11626.918,E2 11626.918} C_VEL
LIN {X 0,Y 517.743,Z 1167.396,A -85,B 0,C 180,E1 11634.854,E2 11634.854} C_VEL
LIN {X 0,Y 524.089,Z 1130.795,A -85,B 0,C 180,E1 11643.123,E2 11643.123} C_VEL
LIN {X 0,Y 535.407,Z 1079.461,A -85,B 0,C 180,E1 11650.835,E2 11650.835} C_VEL
LIN {X 0,Y 549.311,Z 1018.385,A -85,B 0,C 180,E1 11657.022,E2 11657.022} C_VEL
LIN {X 0,Y 563.647,Z 948.629,A -85,B 0,C 180,E1 11661.666,E2 11661.666} C_VEL
LIN {X 0,Y 574.425,Z 878.666,A -85,B 0,C 180,E1 11664.567,E2 11664.567} C_VEL
LIN {X 0,Y 574.22,Z 866.305,A -85,B 0,C 180,E1 11665.148,E2 11665.148} C_VEL
LIN {X 0,Y 548.546,Z 817.095,A -85,B 0,C 180,E1 11670.435,E2 11670.435} C_VEL
LIN {X 0,Y 517.626,Z 773.691,A -85,B 0,C 180,E1 11677.476,E2 11677.476} C_VEL
LIN {X 0,Y 514.149,Z 767.06,A -85,B 0,C 180,E1 11678.795,E2 11678.795} C_VEL
LIN {X 0,Y 514.973,Z 767.06,A -85,B 0,C 180,E1 11688.945,E2 11688.945} C_VEL
LIN {X 0,Y 514.676,Z 767.06,A -85,B 0,C 180,E1 11699.139,E2 11699.139} C_VEL
LIN {X 0,Y 514.37,Z 767.06,A -85,B 0,C 180,E1 11707.609,E2 11707.609} C_VEL
LIN {X 0,Y 514.028,Z 767.06,A -85,B 0,C 180,E1 11716.496,E2 11716.496} C_VEL
LIN {X 0,Y 513.751,Z 767.06,A -85,B 0,C 180,E1 11725.8,E2 11725.8} C_VEL
LIN {X 0,Y 514.086,Z 769.177,A -85,B 0,C 180,E1 11727.351,E2 11727.351} C_VEL
LIN {X 0,Y 543.839,Z 810.298,A -85,B 0,C 180,E1 11734.393,E2 11734.393} C_VEL
LIN {X 0,Y 572.758,Z 861.319,A -85,B 0,C 180,E1 11740.131,E2 11740.131} C_VEL
LIN {X 0,Y 575.974,Z 872.939,A -85,B 0,C 180,E1 11740.963,E2 11740.963} C_VEL
LIN {X 0,Y 565.824,Z 943.082,A -85,B 0,C 180,E1 11743.553,E2 11743.553} C_VEL
LIN {X 0,Y 551.936,Z 1014.514,A -85,B 0,C 180,E1 11747.906,E2 11747.906} C_VEL
LIN {X 0,Y 537.883,Z 1078.11,A -85,B 0,C 180,E1 11753.832,E2 11753.832} C_VEL
LIN {X 0,Y 526.274,Z 1131.126,A -85,B 0,C 180,E1 11761.139,E2 11761.139} C_VEL
LIN {X 0,Y 521.965,Z 1150.919,A -85,B 0,C 180,E1 11764.778,E2 11764.778} C_VEL
LIN {X 0,Y 511.875,Z 1167.289,A -85,B 0,C 180,E1 11768.1,E2 11768.1} C_VEL
LIN {X 0,Y 507.956,Z 1193.914,A -85,B 0,C 180,E1 11776.444,E2 11776.444} C_VEL
LIN {X 0,Y 507.035,Z 1206.763,A -85,B 0,C 180,E1 11783.989,E2 11783.989} C_VEL
LIN {X 0,Y 506.719,Z 1209.837,A -85,B 0,C 180,E1 11790.855,E2 11790.855} C_VEL
LIN {X 0,Y 507.473,Z 1203.491,A -85,B 0,C 180,E1 11798.59,E2 11798.59} C_VEL
LIN {X 0,Y 509.209,Z 1184.079,A -85,B 0,C 180,E1 11807.136,E2 11807.136} C_VEL
LIN {X 0,Y 514.145,Z 1152.377,A -85,B 0,C 180,E1 11815.317,E2 11815.317} C_VEL
LIN {X 0,Y 524.257,Z 1106.239,A -85,B 0,C 180,E1 11823.15,E2 11823.15} C_VEL
LIN {X 0,Y 538.46,Z 1046.95,A -85,B 0,C 180,E1 11829.926,E2 11829.926} C_VEL
LIN {X 0,Y 553.3,Z 979.149,A -85,B 0,C 180,E1 11835.072,E2 11835.072} C_VEL
LIN {X 0,Y 565.732,Z 903.463,A -85,B 0,C 180,E1 11838.678,E2 11838.678} C_VEL
LIN {X 0,Y 568.842,Z 869.938,A -85,B 0,C 180,E1 11839.818,E2 11839.818} C_VEL
LIN {X 0,Y 533.023,Z 807.223,A -85,B 0,C 180,E1 11846.314,E2 11846.314} C_VEL
LIN {X 0,Y 505.975,Z 767.06,A -85,B 0,C 180,E1 11852.141,E2 11852.141} C_VEL
LIN {X 0,Y 506.089,Z 767.06,A -85,B 0,C 180,E1 11861.675,E2 11861.675} C_VEL
LIN {X 0,Y 506.475,Z 767.06,A -85,B 0,C 180,E1 11870.536,E2 11870.536} C_VEL
LIN {X 0,Y 506.67,Z 767.06,A -85,B 0,C 180,E1 11879.159,E2 11879.159} C_VEL
LIN {X 0,Y 506.429,Z 767.06,A -85,B 0,C 180,E1 11887.763,E2 11887.763} C_VEL
LIN {X 0,Y 506.035,Z 767.06,A -85,B 0,C 180,E1 11896.563,E2 11896.563} C_VEL
LIN {X 0,Y 505.724,Z 767.06,A -85,B 0,C 180,E1 11905.799,E2 11905.799} C_VEL
LIN {X 0,Y 505.743,Z 768.941,A -85,B 0,C 180,E1 11914.26,E2 11914.26} C_VEL
LIN {X 0,Y 544.277,Z 825.617,A -85,B 0,C 180,E1 11921.863,E2 11921.863} C_VEL
LIN {X 0,Y 568.848,Z 874.031,A -85,B 0,C 180,E1 11926.638,E2 11926.638} C_VEL
LIN {X 0,Y 558.266,Z 945.786,A -85,B 0,C 180,E1 11929.517,E2 11929.517} C_VEL
LIN {X 0,Y 544.537,Z 1012.779,A -85,B 0,C 180,E1 11933.852,E2 11933.852} C_VEL
LIN {X 0,Y 529.712,Z 1074.62,A -85,B 0,C 180,E1 11939.937,E2 11939.937} C_VEL
LIN {X 0,Y 517.438,Z 1126.709,A -85,B 0,C 180,E1 11947.597,E2 11947.597} C_VEL
LIN {X 0,Y 510.316,Z 1164.145,A -85,B 0,C 180,E1 11955.811,E2 11955.811} C_VEL
LIN {X 0,Y 507.66,Z 1187.452,A -85,B 0,C 180,E1 11964.001,E2 11964.001} C_VEL
LIN {X 0,Y 507.331,Z 1198.911,A -85,B 0,C 180,E1 11972.572,E2 11972.572} C_VEL
LIN {X 0,Y 506.963,Z 1197.516,A -85,B 0,C 180,E1 11981.214,E2 11981.214} C_VEL
LIN {X 0,Y 508.119,Z 1184.782,A -85,B 0,C 180,E1 11989.113,E2 11989.113} C_VEL
LIN {X 0,Y 511.872,Z 1157.518,A -85,B 0,C 180,E1 11997.797,E2 11997.797} C_VEL
LIN {X 0,Y 520.282,Z 1114.955,A -85,B 0,C 180,E1 12006.316,E2 12006.316} C_VEL
LIN {X 0,Y 533.224,Z 1060.725,A -85,B 0,C 180,E1 12013.557,E2 12013.557} C_VEL
LIN {X 0,Y 548.266,Z 995.83,A -85,B 0,C 180,E1 12019.368,E2 12019.368} C_VEL
LIN {X 0,Y 562.589,Z 922.559,A -85,B 0,C 180,E1 12023.58,E2 12023.58} C_VEL
LIN {X 0,Y 569.016,Z 870.727,A -85,B 0,C 180,E1 12025.593,E2 12025.593} C_VEL
LIN {X 0,Y 544.998,Z 823.203,A -85,B 0,C 180,E1 12030.834,E2 12030.834} C_VEL
LIN {X 0,Y 514.787,Z 780.499,A -85,B 0,C 180,E1 12037.915,E2 12037.915} C_VEL
LIN {X 0,Y 506.119,Z 767.06,A -85,B 0,C 180,E1 12040.71,E2 12040.71} C_VEL
LIN {X 0,Y 506.953,Z 767.06,A -85,B 0,C 180,E1 12048.768,E2 12048.768} C_VEL
LIN {X 0,Y 506.679,Z 767.06,A -85,B 0,C 180,E1 12059.125,E2 12059.125} C_VEL
LIN {X 0,Y 506.358,Z 767.06,A -85,B 0,C 180,E1 12067.73,E2 12067.73} C_VEL
LIN {X 0,Y 506.033,Z 767.06,A -85,B 0,C 180,E1 12076.527,E2 12076.527} C_VEL
LIN {X 0,Y 505.945,Z 768.758,A -85,B 0,C 180,E1 12085.272,E2 12085.272} C_VEL
LIN {X 0,Y 535.216,Z 808.406,A -85,B 0,C 180,E1 12092.852,E2 12092.852} C_VEL
LIN {X 0,Y 564.873,Z 859.45,A -85,B 0,C 180,E1 12099.046,E2 12099.046} C_VEL
LIN {X 0,Y 570.61,Z 875.201,A -85,B 0,C 180,E1 12100.401,E2 12100.401} C_VEL
LIN {X 0,Y 559.918,Z 945.42,A -85,B 0,C 180,E1 12103.052,E2 12103.052} C_VEL
LIN {X 0,Y 545.442,Z 1016.138,A -85,B 0,C 180,E1 12107.449,E2 12107.449} C_VEL
LIN {X 0,Y 530.712,Z 1079.782,A -85,B 0,C 180,E1 12113.499,E2 12113.499} C_VEL
LIN {X 0,Y 518.666,Z 1132.409,A -85,B 0,C 180,E1 12120.914,E2 12120.914} C_VEL
LIN {X 0,Y 511.875,Z 1167.289,A -85,B 0,C 180,E1 12128.1,E2 12128.1} C_VEL
LIN {X 0,Y 501.524,Z 1181.163,A -85,B 0,C 180,E1 12131.606,E2 12131.606} C_VEL
LIN {X 0,Y 499.551,Z 1202.149,A -85,B 0,C 180,E1 12140.386,E2 12140.386} C_VEL
LIN {X 0,Y 499.297,Z 1209.395,A -85,B 0,C 180,E1 12147.386,E2 12147.386} C_VEL
LIN {X 0,Y 499.24,Z 1208.366,A -85,B 0,C 180,E1 12154.353,E2 12154.353} C_VEL
LIN {X 0,Y 499.616,Z 1197.202,A -85,B 0,C 180,E1 12162.264,E2 12162.264} C_VEL
LIN {X 0,Y 502.545,Z 1174.69,A -85,B 0,C 180,E1 12170.302,E2 12170.302} C_VEL
LIN {X 0,Y 510.015,Z 1137.069,A -85,B 0,C 180,E1 12178.709,E2 12178.709} C_VEL
LIN {X 0,Y 522.724,Z 1084.509,A -85,B 0,C 180,E1 12186.49,E2 12186.49} C_VEL
LIN {X 0,Y 537.997,Z 1022.313,A -85,B 0,C 180,E1 12192.65,E2 12192.65} C_VEL
LIN {X 0,Y 552.598,Z 953.245,A -85,B 0,C 180,E1 12197.106,E2 12197.106} C_VEL
LIN {X 0,Y 563.332,Z 882.565,A -85,B 0,C 180,E1 12199.924,E2 12199.924} C_VEL
LIN {X 0,Y 562.537,Z 872.525,A -85,B 0,C 180,E1 12200.445,E2 12200.445} C_VEL
LIN {X 0,Y 528.173,Z 811.434,A -85,B 0,C 180,E1 12206.95,E2 12206.95} C_VEL
LIN {X 0,Y 497.905,Z 767.06,A -85,B 0,C 180,E1 12213.805,E2 12213.805} C_VEL
LIN {X 0,Y 498.122,Z 767.06,A -85,B 0,C 180,E1 12223.521,E2 12223.521} C_VEL
LIN {X 0,Y 498.329,Z 767.06,A -85,B 0,C 180,E1 12232.145,E2 12232.145} C_VEL
LIN {X 0,Y 498.672,Z 767.06,A -85,B 0,C 180,E1 12239.146,E2 12239.146} C_VEL
LIN {X 0,Y 498.408,Z 767.06,A -85,B 0,C 180,E1 12247.889,E2 12247.889} C_VEL
LIN {X 0,Y 498.011,Z 767.06,A -85,B 0,C 180,E1 12256.838,E2 12256.838} C_VEL
LIN {X 0,Y 497.694,Z 767.06,A -85,B 0,C 180,E1 12266.246,E2 12266.246} C_VEL
LIN {X 0,Y 497.703,Z 768.782,A -85,B 0,C 180,E1 12272.656,E2 12272.656} C_VEL
LIN {X 0,Y 534.85,Z 822.679,A -85,B 0,C 180,E1 12280.467,E2 12280.467} C_VEL
LIN {X 0,Y 563.186,Z 876.467,A -85,B 0,C 180,E1 12286.101,E2 12286.101} C_VEL
LIN {X 0,Y 552.054,Z 948.527,A -85,B 0,C 180,E1 12289.059,E2 12289.059} C_VEL
LIN {X 0,Y 537.868,Z 1015.006,A -85,B 0,C 180,E1 12293.446,E2 12293.446} C_VEL
LIN {X 0,Y 522.74,Z 1075.465,A -85,B 0,C 180,E1 12299.494,E2 12299.494} C_VEL
LIN {X 0,Y 510.255,Z 1126.289,A -85,B 0,C 180,E1 12307.059,E2 12307.059} C_VEL
LIN {X 0,Y 502.504,Z 1164.481,A -85,B 0,C 180,E1 12315.586,E2 12315.586} C_VEL
LIN {X 0,Y 499.709,Z 1185.769,A -85,B 0,C 180,E1 12323.03,E2 12323.03} C_VEL
LIN {X 0,Y 499.161,Z 1197.769,A -85,B 0,C 180,E1 12330.873,E2 12330.873} C_VEL
LIN {X 0,Y 498.889,Z 1198.77,A -85,B 0,C 180,E1 12339.627,E2 12339.627} C_VEL
LIN {X 0,Y 499.587,Z 1188.379,A -85,B 0,C 180,E1 12347.672,E2 12347.672} C_VEL
LIN {X 0,Y 502.839,Z 1164.574,A -85,B 0,C 180,E1 12356.282,E2 12356.282} C_VEL
LIN {X 0,Y 510.97,Z 1124.552,A -85,B 0,C 180,E1 12365.155,E2 12365.155} C_VEL
LIN {X 0,Y 523.447,Z 1073.349,A -85,B 0,C 180,E1 12372.668,E2 12372.668} C_VEL
LIN {X 0,Y 539.09,Z 1009.484,A -85,B 0,C 180,E1 12378.946,E2 12378.946} C_VEL
LIN {X 0,Y 554.514,Z 938.555,A -85,B 0,C 180,E1 12383.443,E2 12383.443} C_VEL
LIN {X 0,Y 563.625,Z 874.43,A -85,B 0,C 180,E1 12386.109,E2 12386.109} C_VEL
LIN {X 0,Y 539.747,Z 826.339,A -85,B 0,C 180,E1 12391.615,E2 12391.615} C_VEL
LIN {X 0,Y 508.312,Z 781.572,A -85,B 0,C 180,E1 12399.456,E2 12399.456} C_VEL
LIN {X 0,Y 498.328,Z 767.06,A -85,B 0,C 180,E1 12403.174,E2 12403.174} C_VEL
LIN {X 0,Y 498.448,Z 767.06,A -85,B 0,C 180,E1 12412.111,E2 12412.111} C_VEL
LIN {X 0,Y 498.68,Z 767.06,A -85,B 0,C 180,E1 12419.111,E2 12419.111} C_VEL
LIN {X 0,Y 498.334,Z 767.06,A -85,B 0,C 180,E1 12427.855,E2 12427.855} C_VEL
LIN {X 0,Y 498.003,Z 767.06,A -85,B 0,C 180,E1 12436.801,E2 12436.801} C_VEL
LIN {X 0,Y 498.004,Z 768.728,A -85,B 0,C 180,E1 12442.986,E2 12442.986} C_VEL
LIN {X 0,Y 524.273,Z 803.756,A -85,B 0,C 180,E1 12450.636,E2 12450.636} C_VEL
LIN {X 0,Y 552.573,Z 849.267,A -85,B 0,C 180,E1 12456.947,E2 12456.947} C_VEL
LIN {X 0,Y 565.027,Z 879.501,A -85,B 0,C 180,E1 12459.899,E2 12459.899} C_VEL
LIN {X 0,Y 553.967,Z 948.285,A -85,B 0,C 180,E1 12462.562,E2 12462.562} C_VEL
LIN {X 0,Y 538.82,Z 1018.86,A -85,B 0,C 180,E1 12467.065,E2 12467.065} C_VEL
LIN {X 0,Y 523.28,Z 1082.661,A -85,B 0,C 180,E1 12473.296,E2 12473.296} C_VEL
LIN {X 0,Y 510.514,Z 1135.651,A -85,B 0,C 180,E1 12481.039,E2 12481.039} C_VEL
LIN {X 0,Y 502.906,Z 1173.253,A -85,B 0,C 180,E1 12489.284,E2 12489.284} C_VEL
LIN {X 0,Y 501.524,Z 1181.163,A -85,B 0,C 180,E1 12491.606,E2 12491.606} C_VEL
LIN {X 0,Y 492.51,Z 1192.357,A -85,B 0,C 180,E1 12495.368,E2 12495.368} C_VEL
LIN {X 0,Y 491.075,Z 1206.757,A -85,B 0,C 180,E1 12503.793,E2 12503.793} C_VEL
LIN {X 0,Y 490.732,Z 1209.837,A -85,B 0,C 180,E1 12510.883,E2 12510.883} C_VEL
LIN {X 0,Y 491.502,Z 1203.76,A -85,B 0,C 180,E1 12518.669,E2 12518.669} C_VEL
LIN {X 0,Y 493.335,Z 1184.74,A -85,B 0,C 180,E1 12527.477,E2 12527.477} C_VEL
LIN {X 0,Y 499.064,Z 1152.275,A -85,B 0,C 180,E1 12536.139,E2 12536.139} C_VEL
LIN {X 0,Y 510.25,Z 1105.953,A -85,B 0,C 180,E1 12544.197,E2 12544.197} C_VEL
LIN {X 0,Y 525.726,Z 1046.772,A -85,B 0,C 180,E1 12551.089,E2 12551.089} C_VEL
LIN {X 0,Y 541.597,Z 979.094,A -85,B 0,C 180,E1 12556.27,E2 12556.27} C_VEL
LIN {X 0,Y 554.792,Z 903.729,A -85,B 0,C 180,E1 12559.891,E2 12559.891} C_VEL
LIN {X 0,Y 557.347,Z 877.194,A -85,B 0,C 180,E1 12560.859,E2 12560.859} C_VEL
LIN {X 0,Y 524.253,Z 817.144,A -85,B 0,C 180,E1 12567.412,E2 12567.412} C_VEL
LIN {X 0,Y 492.651,Z 773.11,A -85,B 0,C 180,E1 12574.392,E2 12574.392} C_VEL
LIN {X 0,Y 489.829,Z 767.06,A -85,B 0,C 180,E1 12575.308,E2 12575.308} C_VEL
LIN {X 0,Y 490.105,Z 767.06,A -85,B 0,C 180,E1 12584.766,E2 12584.766} C_VEL
LIN {X 0,Y 490.381,Z 767.06,A -85,B 0,C 180,E1 12593.803,E2 12593.803} C_VEL
LIN {X 0,Y 490.508,Z 767.06,A -85,B 0,C 180,E1 12600.904,E2 12600.904} C_VEL
LIN {X 0,Y 490.346,Z 767.06,A -85,B 0,C 180,E1 12609.814,E2 12609.814} C_VEL
LIN {X 0,Y 489.901,Z 767.06,A -85,B 0,C 180,E1 12619.255,E2 12619.255} C_VEL
LIN {X 0,Y 489.64,Z 767.06,A -85,B 0,C 180,E1 12628.717,E2 12628.717} C_VEL
LIN {X 0,Y 489.753,Z 768.814,A -85,B 0,C 180,E1 12630.939,E2 12630.939} C_VEL
LIN {X 0,Y 525.551,Z 820.052,A -85,B 0,C 180,E1 12639.005,E2 12639.005} C_VEL
LIN {X 0,Y 557.107,Z 878.101,A -85,B 0,C 180,E1 12645.465,E2 12645.465} C_VEL
LIN {X 0,Y 545.443,Z 953.349,A -85,B 0,C 180,E1 12648.704,E2 12648.704} C_VEL
LIN {X 0,Y 530.374,Z 1020.418,A -85,B 0,C 180,E1 12653.303,E2 12653.303} C_VEL
LIN {X 0,Y 514.461,Z 1081.353,A -85,B 0,C 180,E1 12659.686,E2 12659.686} C_VEL
LIN {X 0,Y 501.597,Z 1131.498,A -85,B 0,C 180,E1 12667.574,E2 12667.574} C_VEL
LIN {X 0,Y 494.218,Z 1167.856,A -85,B 0,C 180,E1 12676.261,E2 12676.261} C_VEL
LIN {X 0,Y 491.772,Z 1189.545,A -85,B 0,C 180,E1 12684.695,E2 12684.695} C_VEL
LIN {X 0,Y 491.319,Z 1199.018,A -85,B 0,C 180,E1 12692.656,E2 12692.656} C_VEL
LIN {X 0,Y 490.977,Z 1197.318,A -85,B 0,C 180,E1 12701.584,E2 12701.584} C_VEL
LIN {X 0,Y 492.512,Z 1183.78,A -85,B 0,C 180,E1 12710.006,E2 12710.006} C_VEL
LIN {X 0,Y 496.738,Z 1154.944,A -85,B 0,C 180,E1 12719.201,E2 12719.201} C_VEL
LIN {X 0,Y 506.657,Z 1111.682,A -85,B 0,C 180,E1 12727.852,E2 12727.852} C_VEL
LIN {X 0,Y 520.993,Z 1057.262,A -85,B 0,C 180,E1 12735.081,E2 12735.081} C_VEL
LIN {X 0,Y 537.574,Z 992.002,A -85,B 0,C 180,E1 12740.877,E2 12740.877} C_VEL
LIN {X 0,Y 552.365,Z 920.737,A -85,B 0,C 180,E1 12744.948,E2 12744.948} C_VEL
LIN {X 0,Y 558.06,Z 877.544,A -85,B 0,C 180,E1 12746.695,E2 12746.695} C_VEL
LIN {X 0,Y 535.229,Z 831.179,A -85,B 0,C 180,E1 12752.217,E2 12752.217} C_VEL
LIN {X 0,Y 505.947,Z 788.816,A -85,B 0,C 180,E1 12759.814,E2 12759.814} C_VEL
LIN {X 0,Y 490.681,Z 767.06,A -85,B 0,C 180,E1 12765.664,E2 12765.664} C_VEL
LIN {X 0,Y 490.825,Z 767.06,A -85,B 0,C 180,E1 12775.551,E2 12775.551} C_VEL
LIN {X 0,Y 490.63,Z 767.06,A -85,B 0,C 180,E1 12786.194,E2 12786.194} C_VEL
LIN {X 0,Y 490.137,Z 767.06,A -85,B 0,C 180,E1 12795.233,E2 12795.233} C_VEL
LIN {X 0,Y 490.227,Z 769.049,A -85,B 0,C 180,E1 12800.403,E2 12800.403} C_VEL
LIN {X 0,Y 512.807,Z 798.571,A -85,B 0,C 180,E1 12807.994,E2 12807.994} C_VEL
LIN {X 0,Y 541.291,Z 841.643,A -85,B 0,C 180,E1 12814.92,E2 12814.92} C_VEL
LIN {X 0,Y 559.687,Z 881.881,A -85,B 0,C 180,E1 12819.319,E2 12819.319} C_VEL
LIN {X 0,Y 548.051,Z 951.312,A -85,B 0,C 180,E1 12822.073,E2 12822.073} C_VEL
LIN {X 0,Y 532.163,Z 1021.644,A -85,B 0,C 180,E1 12826.67,E2 12826.67} C_VEL
LIN {X 0,Y 516.083,Z 1084.317,A -85,B 0,C 180,E1 12832.957,E2 12832.957} C_VEL
LIN {X 0,Y 503.196,Z 1135.547,A -85,B 0,C 180,E1 12840.576,E2 12840.576} C_VEL
LIN {X 0,Y 494.877,Z 1174.672,A -85,B 0,C 180,E1 12849.363,E2 12849.363} C_VEL
LIN {X 0,Y 492.51,Z 1192.357,A -85,B 0,C 180,E1 12855.368,E2 12855.368} C_VEL
LIN {X 0,Y 483.488,Z 1200.787,A -85,B 0,C 180,E1 12859.273,E2 12859.273} C_VEL
LIN {X 0,Y 483.278,Z 1209.389,A -85,B 0,C 180,E1 12867.3,E2 12867.3} C_VEL
LIN {X 0,Y 483.219,Z 1208.36,A -85,B 0,C 180,E1 12874.497,E2 12874.497} C_VEL
LIN {X 0,Y 483.719,Z 1197.196,A -85,B 0,C 180,E1 12882.674,E2 12882.674} C_VEL
LIN {X 0,Y 487.315,Z 1173.835,A -85,B 0,C 180,E1 12891.223,E2 12891.223} C_VEL
LIN {X 0,Y 496.484,Z 1133.489,A -85,B 0,C 180,E1 12900.26,E2 12900.26} C_VEL
LIN {X 0,Y 510.407,Z 1080.474,A -85,B 0,C 180,E1 12908.071,E2 12908.071} C_VEL
LIN {X 0,Y 526.67,Z 1018.203,A -85,B 0,C 180,E1 12914.165,E2 12914.165} C_VEL
LIN {X 0,Y 542.162,Z 948.527,A -85,B 0,C 180,E1 12918.577,E2 12918.577} C_VEL
LIN {X 0,Y 551.618,Z 880.632,A -85,B 0,C 180,E1 12921.389,E2 12921.389} C_VEL
LIN {X 0,Y 519.639,Z 821.791,A -85,B 0,C 180,E1 12928.015,E2 12928.015} C_VEL
LIN {X 0,Y 489.004,Z 778.938,A -85,B 0,C 180,E1 12935.018,E2 12935.018} C_VEL
LIN {X 0,Y 481.851,Z 767.06,A -85,B 0,C 180,E1 12937.209,E2 12937.209} C_VEL
LIN {X 0,Y 482.17,Z 767.06,A -85,B 0,C 180,E1 12946.371,E2 12946.371} C_VEL
LIN {X 0,Y 483.091,Z 767.06,A -85,B 0,C 180,E1 12957.318,E2 12957.318} C_VEL
LIN {X 0,Y 482.661,Z 767.06,A -85,B 0,C 180,E1 12966.333,E2 12966.333} C_VEL
LIN {X 0,Y 481.996,Z 767.06,A -85,B 0,C 180,E1 12976.353,E2 12976.353} C_VEL
LIN {X 0,Y 481.596,Z 767.06,A -85,B 0,C 180,E1 12986.186,E2 12986.186} C_VEL
LIN {X 0,Y 481.795,Z 768.83,A -85,B 0,C 180,E1 12989.057,E2 12989.057} C_VEL
LIN {X 0,Y 515.114,Z 815.676,A -85,B 0,C 180,E1 12997.195,E2 12997.195} C_VEL
LIN {X 0,Y 546.431,Z 871.081,A -85,B 0,C 180,E1 13003.831,E2 13003.831} C_VEL
LIN {X 0,Y 551.403,Z 885.982,A -85,B 0,C 180,E1 13005.142,E2 13005.142} C_VEL
LIN {X 0,Y 538.313,Z 960.721,A -85,B 0,C 180,E1 13008.478,E2 13008.478} C_VEL
LIN {X 0,Y 522.396,Z 1028,A -85,B 0,C 180,E1 13013.351,E2 13013.351} C_VEL
LIN {X 0,Y 506.134,Z 1087.244,A -85,B 0,C 180,E1 13019.88,E2 13019.88} C_VEL
LIN {X 0,Y 493.307,Z 1135.529,A -85,B 0,C 180,E1 13027.881,E2 13027.881} C_VEL
LIN {X 0,Y 486.159,Z 1169.638,A -85,B 0,C 180,E1 13036.473,E2 13036.473} C_VEL
LIN {X 0,Y 483.849,Z 1191.254,A -85,B 0,C 180,E1 13045.509,E2 13045.509} C_VEL
LIN {X 0,Y 483.295,Z 1199.072,A -85,B 0,C 180,E1 13052.7,E2 13052.7} C_VEL
LIN {X 0,Y 482.997,Z 1197.219,A -85,B 0,C 180,E1 13061.778,E2 13061.778} C_VEL
LIN {X 0,Y 484.595,Z 1183.541,A -85,B 0,C 180,E1 13070.347,E2 13070.347} C_VEL
LIN {X 0,Y 489.136,Z 1154.581,A -85,B 0,C 180,E1 13079.7,E2 13079.7} C_VEL
LIN {X 0,Y 499.246,Z 1112.999,A -85,B 0,C 180,E1 13088.164,E2 13088.164} C_VEL
LIN {X 0,Y 514.547,Z 1057.429,A -85,B 0,C 180,E1 13095.671,E2 13095.671} C_VEL
LIN {X 0,Y 531.789,Z 992.642,A -85,B 0,C 180,E1 13101.48,E2 13101.48} C_VEL
LIN {X 0,Y 547.255,Z 920.736,A -85,B 0,C 180,E1 13105.612,E2 13105.612} C_VEL
LIN {X 0,Y 552.789,Z 881.434,A -85,B 0,C 180,E1 13107.225,E2 13107.225} C_VEL
LIN {X 0,Y 530.75,Z 835.86,A -85,B 0,C 180,E1 13112.828,E2 13112.828} C_VEL
LIN {X 0,Y 503.28,Z 795.634,A -85,B 0,C 180,E1 13120.276,E2 13120.276} C_VEL
LIN {X 0,Y 486.076,Z 773.469,A -85,B 0,C 180,E1 13126.758,E2 13126.758} C_VEL
LIN {X 0,Y 482.78,Z 767.06,A -85,B 0,C 180,E1 13129.116,E2 13129.116} C_VEL
LIN {X 0,Y 482.701,Z 767.06,A -85,B 0,C 180,E1 13139.082,E2 13139.082} C_VEL
LIN {X 0,Y 482.316,Z 767.06,A -85,B 0,C 180,E1 13148.118,E2 13148.118} C_VEL
LIN {X 0,Y 482.223,Z 769.084,A -85,B 0,C 180,E1 13157.15,E2 13157.15} C_VEL
LIN {X 0,Y 495.413,Z 786.333,A -85,B 0,C 180,E1 13162.9,E2 13162.9} C_VEL
LIN {X 0,Y 518.861,Z 817.426,A -85,B 0,C 180,E1 13169.932,E2 13169.932} C_VEL
LIN {X 0,Y 544.914,Z 861.928,A -85,B 0,C 180,E1 13176.308,E2 13176.308} C_VEL
LIN {X 0,Y 554.299,Z 885.324,A -85,B 0,C 180,E1 13178.763,E2 13178.763} C_VEL
LIN {X 0,Y 541.974,Z 954.987,A -85,B 0,C 180,E1 13181.623,E2 13181.623} C_VEL
LIN {X 0,Y 525.502,Z 1024.358,A -85,B 0,C 180,E1 13186.275,E2 13186.275} C_VEL
LIN {X 0,Y 508.897,Z 1085.99,A -85,B 0,C 180,E1 13192.613,E2 13192.613} C_VEL
LIN {X 0,Y 495.534,Z 1136.819,A -85,B 0,C 180,E1 13200.362,E2 13200.362} C_VEL
LIN {X 0,Y 487.16,Z 1174.648,A -85,B 0,C 180,E1 13209.021,E2 13209.021} C_VEL
LIN {X 0,Y 483.668,Z 1197.185,A -85,B 0,C 180,E1 13217.319,E2 13217.319} C_VEL
LIN {X 0,Y 483.488,Z 1200.787,A -85,B 0,C 180,E1 13219.273,E2 13219.273} C_VEL
LIN {X 0,Y 475.142,Z 1206.538,A -85,B 0,C 180,E1 13223.36,E2 13223.36} C_VEL
LIN {X 0,Y 474.745,Z 1209.837,A -85,B 0,C 180,E1 13230.912,E2 13230.912} C_VEL
LIN {X 0,Y 475.513,Z 1203.613,A -85,B 0,C 180,E1 13239.071,E2 13239.071} C_VEL
LIN {X 0,Y 477.566,Z 1184.947,A -85,B 0,C 180,E1 13247.989,E2 13247.989} C_VEL
LIN {X 0,Y 484.086,Z 1152.087,A -85,B 0,C 180,E1 13257.012,E2 13257.012} C_VEL
LIN {X 0,Y 496.199,Z 1106.513,A -85,B 0,C 180,E1 13265.181,E2 13265.181} C_VEL
LIN {X 0,Y 512.676,Z 1048.319,A -85,B 0,C 180,E1 13272.122,E2 13272.122} C_VEL
LIN {X 0,Y 529.574,Z 981.381,A -85,B 0,C 180,E1 13277.366,E2 13277.366} C_VEL
LIN {X 0,Y 543.674,Z 906.627,A -85,B 0,C 180,E1 13281.051,E2 13281.051} C_VEL
LIN {X 0,Y 545.797,Z 884.112,A -85,B 0,C 180,E1 13281.943,E2 13281.943} C_VEL
LIN {X 0,Y 515.104,Z 826.233,A -85,B 0,C 180,E1 13288.63,E2 13288.63} C_VEL
LIN {X 0,Y 483.18,Z 781.064,A -85,B 0,C 180,E1 13296.302,E2 13296.302} C_VEL
LIN {X 0,Y 473.845,Z 767.06,A -85,B 0,C 180,E1 13299.402,E2 13299.402} C_VEL
LIN {X 0,Y 474.391,Z 767.06,A -85,B 0,C 180,E1 13309.89,E2 13309.89} C_VEL
LIN {X 0,Y 474.703,Z 767.06,A -85,B 0,C 180,E1 13319.103,E2 13319.103} C_VEL
LIN {X 0,Y 474.361,Z 767.06,A -85,B 0,C 180,E1 13328.292,E2 13328.292} C_VEL
LIN {X 0,Y 473.9,Z 767.06,A -85,B 0,C 180,E1 13337.722,E2 13337.722} C_VEL
LIN {X 0,Y 473.829,Z 768.921,A -85,B 0,C 180,E1 13346.969,E2 13346.969} C_VEL
LIN {X 0,Y 504.095,Z 810.571,A -85,B 0,C 180,E1 13355.089,E2 13355.089} C_VEL
LIN {X 0,Y 535.398,Z 863.597,A -85,B 0,C 180,E1 13362.037,E2 13362.037} C_VEL
LIN {X 0,Y 545.636,Z 889.255,A -85,B 0,C 180,E1 13364.612,E2 13364.612} C_VEL
LIN {X 0,Y 532.226,Z 962.811,A -85,B 0,C 180,E1 13367.969,E2 13367.969} C_VEL
LIN {X 0,Y 515.672,Z 1030.126,A -85,B 0,C 180,E1 13372.929,E2 13372.929} C_VEL
LIN {X 0,Y 498.716,Z 1089.602,A -85,B 0,C 180,E1 13379.637,E2 13379.637} C_VEL
LIN {X 0,Y 485.529,Z 1137.157,A -85,B 0,C 180,E1 13387.75,E2 13387.75} C_VEL
LIN {X 0,Y 478.141,Z 1171.47,A -85,B 0,C 180,E1 13396.709,E2 13396.709} C_VEL
LIN {X 0,Y 475.767,Z 1192.907,A -85,B 0,C 180,E1 13406.348,E2 13406.348} C_VEL
LIN {X 0,Y 474.862,Z 1199.75,A -85,B 0,C 180,E1 13414.582,E2 13414.582} C_VEL
LIN {X 0,Y 475.186,Z 1196.057,A -85,B 0,C 180,E1 13423.114,E2 13423.114} C_VEL
LIN {X 0,Y 476.965,Z 1179.641,A -85,B 0,C 180,E1 13432.191,E2 13432.191} C_VEL
LIN {X 0,Y 482.02,Z 1151.495,A -85,B 0,C 180,E1 13440.887,E2 13440.887} C_VEL
LIN {X 0,Y 493.55,Z 1107.723,A -85,B 0,C 180,E1 13449.553,E2 13449.553} C_VEL
LIN {X 0,Y 510.125,Z 1050.927,A -85,B 0,C 180,E1 13456.996,E2 13456.996} C_VEL
LIN {X 0,Y 527.813,Z 986.499,A -85,B 0,C 180,E1 13462.57,E2 13462.57} C_VEL
LIN {X 0,Y 543.664,Z 913.054,A -85,B 0,C 180,E1 13466.612,E2 13466.612} C_VEL
LIN {X 0,Y 547.374,Z 884.722,A -85,B 0,C 180,E1 13467.824,E2 13467.824} C_VEL
LIN {X 0,Y 525.424,Z 838.959,A -85,B 0,C 180,E1 13473.689,E2 13473.689} C_VEL
LIN {X 0,Y 499.857,Z 801.447,A -85,B 0,C 180,E1 13481,E2 13481} C_VEL
LIN {X 0,Y 483.721,Z 780.384,A -85,B 0,C 180,E1 13487.359,E2 13487.359} C_VEL
LIN {X 0,Y 478.902,Z 774.045,A -85,B 0,C 180,E1 13489.949,E2 13489.949} C_VEL
LIN {X 0,Y 474.445,Z 767.06,A -85,B 0,C 180,E1 13493.557,E2 13493.557} C_VEL
LIN {X 0,Y 474.467,Z 767.06,A -85,B 0,C 180,E1 13500.898,E2 13500.898} C_VEL
LIN {X 0,Y 474.259,Z 767.06,A -85,B 0,C 180,E1 13510.113,E2 13510.113} C_VEL
LIN {X 0,Y 474.55,Z 769.292,A -85,B 0,C 180,E1 13512.977,E2 13512.977} C_VEL
LIN {X 0,Y 481.637,Z 778.86,A -85,B 0,C 180,E1 13517.449,E2 13517.449} C_VEL
LIN {X 0,Y 493.169,Z 793.13,A -85,B 0,C 180,E1 13522.472,E2 13522.472} C_VEL
LIN {X 0,Y 516.613,Z 825.101,A -85,B 0,C 180,E1 13529.722,E2 13529.722} C_VEL
LIN {X 0,Y 541.615,Z 869.448,A -85,B 0,C 180,E1 13536.135,E2 13536.135} C_VEL
LIN {X 0,Y 548.761,Z 890.152,A -85,B 0,C 180,E1 13538.236,E2 13538.236} C_VEL
LIN {X 0,Y 536.079,Z 957.885,A -85,B 0,C 180,E1 13541.114,E2 13541.114} C_VEL
LIN {X 0,Y 518.9,Z 1026.911,A -85,B 0,C 180,E1 13545.851,E2 13545.851} C_VEL
LIN {X 0,Y 501.233,Z 1089.477,A -85,B 0,C 180,E1 13552.489,E2 13552.489} C_VEL
LIN {X 0,Y 487.009,Z 1141.202,A -85,B 0,C 180,E1 13560.739,E2 13560.739} C_VEL
LIN {X 0,Y 478.909,Z 1176.872,A -85,B 0,C 180,E1 13569.371,E2 13569.371} C_VEL
LIN {X 0,Y 475.526,Z 1199.007,A -85,B 0,C 180,E1 13578.034,E2 13578.034} C_VEL
LIN {X 0,Y 475.142,Z 1206.538,A -85,B 0,C 180,E1 13583.36,E2 13583.36} C_VEL
LIN {X 0,Y 467.145,Z 1209.467,A -85,B 0,C 180,E1 13587.552,E2 13587.552} C_VEL
LIN {X 0,Y 467.187,Z 1208.354,A -85,B 0,C 180,E1 13594.652,E2 13594.652} C_VEL
LIN {X 0,Y 467.824,Z 1197.49,A -85,B 0,C 180,E1 13602.959,E2 13602.959} C_VEL
LIN {X 0,Y 472.119,Z 1172.918,A -85,B 0,C 180,E1 13612.171,E2 13612.171} C_VEL
LIN {X 0,Y 482.413,Z 1131.941,A -85,B 0,C 180,E1 13621.508,E2 13621.508} C_VEL
LIN {X 0,Y 497.185,Z 1080.579,A -85,B 0,C 180,E1 13629.204,E2 13629.204} C_VEL
LIN {X 0,Y 514.464,Z 1018.79,A -85,B 0,C 180,E1 13635.356,E2 13635.356} C_VEL
LIN {X 0,Y 531.107,Z 948.51,A -85,B 0,C 180,E1 13639.856,E2 13639.856} C_VEL
LIN {X 0,Y 540.369,Z 888.109,A -85,B 0,C 180,E1 13642.439,E2 13642.439} C_VEL
LIN {X 0,Y 510.632,Z 831.055,A -85,B 0,C 180,E1 13649.244,E2 13649.244} C_VEL
LIN {X 0,Y 480.143,Z 787.645,A -85,B 0,C 180,E1 13656.822,E2 13656.822} C_VEL
LIN {X 0,Y 465.971,Z 767.06,A -85,B 0,C 180,E1 13662.006,E2 13662.006} C_VEL
LIN {X 0,Y 466.316,Z 767.06,A -85,B 0,C 180,E1 13671.602,E2 13671.602} C_VEL
LIN {X 0,Y 466.705,Z 767.06,A -85,B 0,C 180,E1 13679.087,E2 13679.087} C_VEL
LIN {X 0,Y 466.347,Z 767.06,A -85,B 0,C 180,E1 13688.435,E2 13688.435} C_VEL
LIN {X 0,Y 465.874,Z 767.06,A -85,B 0,C 180,E1 13698.038,E2 13698.038} C_VEL
LIN {X 0,Y 465.763,Z 768.829,A -85,B 0,C 180,E1 13704.575,E2 13704.575} C_VEL
LIN {X 0,Y 491.673,Z 803.482,A -85,B 0,C 180,E1 13712.414,E2 13712.414} C_VEL
LIN {X 0,Y 522.877,Z 853.413,A -85,B 0,C 180,E1 13719.791,E2 13719.791} C_VEL
LIN {X 0,Y 539.992,Z 891.963,A -85,B 0,C 180,E1 13724.052,E2 13724.052} C_VEL
LIN {X 0,Y 526.38,Z 963.959,A -85,B 0,C 180,E1 13727.392,E2 13727.392} C_VEL
LIN {X 0,Y 509.331,Z 1030.99,A -85,B 0,C 180,E1 13732.388,E2 13732.388} C_VEL
LIN {X 0,Y 491.79,Z 1090.328,A -85,B 0,C 180,E1 13739.163,E2 13739.163} C_VEL
LIN {X 0,Y 478.028,Z 1137.789,A -85,B 0,C 180,E1 13747.398,E2 13747.398} C_VEL
LIN {X 0,Y 470.284,Z 1171.847,A -85,B 0,C 180,E1 13756.483,E2 13756.483} C_VEL
LIN {X 0,Y 467.799,Z 1193.037,A -85,B 0,C 180,E1 13766.285,E2 13766.285} C_VEL
LIN {X 0,Y 466.848,Z 1199.769,A -85,B 0,C 180,E1 13774.661,E2 13774.661} C_VEL
LIN {X 0,Y 467.219,Z 1195.957,A -85,B 0,C 180,E1 13783.342,E2 13783.342} C_VEL
LIN {X 0,Y 469.118,Z 1178.943,A -85,B 0,C 180,E1 13792.802,E2 13792.802} C_VEL
LIN {X 0,Y 474.564,Z 1151.011,A -85,B 0,C 180,E1 13801.457,E2 13801.457} C_VEL
LIN {X 0,Y 486.757,Z 1107.218,A -85,B 0,C 180,E1 13810.2,E2 13810.2} C_VEL
LIN {X 0,Y 504.2,Z 1050.374,A -85,B 0,C 180,E1 13817.703,E2 13817.703} C_VEL
LIN {X 0,Y 522.235,Z 987.12,A -85,B 0,C 180,E1 13823.207,E2 13823.207} C_VEL
LIN {X 0,Y 538.476,Z 914.601,A -85,B 0,C 180,E1 13827.237,E2 13827.237} C_VEL
LIN {X 0,Y 542.089,Z 888.336,A -85,B 0,C 180,E1 13828.394,E2 13828.394} C_VEL
LIN {X 0,Y 521.08,Z 843.772,A -85,B 0,C 180,E1 13834.323,E2 13834.323} C_VEL
LIN {X 0,Y 494.977,Z 804.23,A -85,B 0,C 180,E1 13842.309,E2 13842.309} C_VEL
LIN {X 0,Y 478.139,Z 782.14,A -85,B 0,C 180,E1 13849.818,E2 13849.818} C_VEL
LIN {X 0,Y 470.446,Z 773.776,A -85,B 0,C 180,E1 13855.59,E2 13855.59} C_VEL
LIN {X 0,Y 467.468,Z 770.605,A -85,B 0,C 180,E1 13865.568,E2 13865.568} C_VEL
LIN {X 0,Y 473.47,Z 777.611,A -85,B 0,C 180,E1 13872.95,E2 13872.95} C_VEL
LIN {X 0,Y 485.162,Z 792.13,A -85,B 0,C 180,E1 13879.62,E2 13879.62} C_VEL
LIN {X 0,Y 508.957,Z 824.265,A -85,B 0,C 180,E1 13887.977,E2 13887.977} C_VEL
LIN {X 0,Y 534.044,Z 867.976,A -85,B 0,C 180,E1 13894.85,E2 13894.85} C_VEL
LIN {X 0,Y 543.559,Z 893.255,A -85,B 0,C 180,E1 13897.649,E2 13897.649} C_VEL
LIN {X 0,Y 529.92,Z 962.277,A -85,B 0,C 180,E1 13900.678,E2 13900.678} C_VEL
LIN {X 0,Y 512.099,Z 1030.446,A -85,B 0,C 180,E1 13905.504,E2 13905.504} C_VEL
LIN {X 0,Y 494.108,Z 1091.25,A -85,B 0,C 180,E1 13912.131,E2 13912.131} C_VEL
LIN {X 0,Y 479.517,Z 1141.911,A -85,B 0,C 180,E1 13920.411,E2 13920.411} C_VEL
LIN {X 0,Y 470.843,Z 1178.293,A -85,B 0,C 180,E1 13929.484,E2 13929.484} C_VEL
LIN {X 0,Y 467.589,Z 1199.004,A -85,B 0,C 180,E1 13937.828,E2 13937.828} C_VEL
LIN {X 0,Y 467.142,Z 1208.35,A -85,B 0,C 180,E1 13945.342,E2 13945.342} C_VEL
LIN {X 0,Y 467.145,Z 1209.467,A -85,B 0,C 180,E1 13947.552,E2 13947.552} C_VEL
LIN {X 0,Y 458.875,Z 1209.63,A -85,B 0,C 180,E1 13951.81,E2 13951.81} C_VEL
LIN {X 0,Y 459.609,Z 1202.093,A -85,B 0,C 180,E1 13960.453,E2 13960.453} C_VEL
LIN {X 0,Y 462.268,Z 1181.941,A -85,B 0,C 180,E1 13969.646,E2 13969.646} C_VEL
LIN {X 0,Y 470.067,Z 1148.614,A -85,B 0,C 180,E1 13978.674,E2 13978.674} C_VEL
LIN {X 0,Y 484.226,Z 1100.702,A -85,B 0,C 180,E1 13987.134,E2 13987.134} C_VEL
LIN {X 0,Y 502.095,Z 1041.601,A -85,B 0,C 180,E1 13993.997,E2 13993.997} C_VEL
LIN {X 0,Y 519.825,Z 974.567,A -85,B 0,C 180,E1 13999.072,E2 13999.072} C_VEL
LIN {X 0,Y 534.288,Z 900.753,A -85,B 0,C 180,E1 14002.556,E2 14002.556} C_VEL
LIN {X 0,Y 534.082,Z 890.304,A -85,B 0,C 180,E1 14003.152,E2 14003.152} C_VEL
LIN {X 0,Y 505.892,Z 835.401,A -85,B 0,C 180,E1 14009.924,E2 14009.924} C_VEL
LIN {X 0,Y 477.16,Z 794.098,A -85,B 0,C 180,E1 14017.348,E2 14017.348} C_VEL
LIN {X 0,Y 460.537,Z 772.971,A -85,B 0,C 180,E1 14023.085,E2 14023.085} C_VEL
LIN {X 0,Y 457.996,Z 767.06,A -85,B 0,C 180,E1 14024.655,E2 14024.655} C_VEL
LIN {X 0,Y 458.675,Z 767.06,A -85,B 0,C 180,E1 14035.277,E2 14035.277} C_VEL
LIN {X 0,Y 458.859,Z 767.06,A -85,B 0,C 180,E1 14044.76,E2 14044.76} C_VEL
LIN {X 0,Y 458.115,Z 767.06,A -85,B 0,C 180,E1 14054.398,E2 14054.398} C_VEL
LIN {X 0,Y 457.93,Z 768.79,A -85,B 0,C 180,E1 14061.886,E2 14061.886} C_VEL
LIN {X 0,Y 480.336,Z 798.529,A -85,B 0,C 180,E1 14069.695,E2 14069.695} C_VEL
LIN {X 0,Y 510.073,Z 843.716,A -85,B 0,C 180,E1 14077.323,E2 14077.323} C_VEL
LIN {X 0,Y 534.517,Z 893.168,A -85,B 0,C 180,E1 14083.412,E2 14083.412} C_VEL
LIN {X 0,Y 520.114,Z 967.022,A -85,B 0,C 180,E1 14086.922,E2 14086.922} C_VEL
LIN {X 0,Y 502.659,Z 1032.952,A -85,B 0,C 180,E1 14091.937,E2 14091.937} C_VEL
LIN {X 0,Y 484.865,Z 1091.016,A -85,B 0,C 180,E1 14098.673,E2 14098.673} C_VEL
LIN {X 0,Y 470.791,Z 1137.555,A -85,B 0,C 180,E1 14106.841,E2 14106.841} C_VEL
LIN {X 0,Y 462.67,Z 1170.891,A -85,B 0,C 180,E1 14115.772,E2 14115.772} C_VEL
LIN {X 0,Y 459.849,Z 1191.818,A -85,B 0,C 180,E1 14125.274,E2 14125.274} C_VEL
LIN {X 0,Y 459.251,Z 1199.233,A -85,B 0,C 180,E1 14132.842,E2 14132.842} C_VEL
LIN {X 0,Y 458.885,Z 1198.47,A -85,B 0,C 180,E1 14140.475,E2 14140.475} C_VEL
LIN {X 0,Y 460.165,Z 1187.494,A -85,B 0,C 180,E1 14149.187,E2 14149.187} C_VEL
LIN {X 0,Y 464.781,Z 1162.508,A -85,B 0,C 180,E1 14158.769,E2 14158.769} C_VEL
LIN {X 0,Y 475.455,Z 1122.541,A -85,B 0,C 180,E1 14168.082,E2 14168.082} C_VEL
LIN {X 0,Y 492.265,Z 1069.242,A -85,B 0,C 180,E1 14176.187,E2 14176.187} C_VEL
LIN {X 0,Y 511.312,Z 1006.594,A -85,B 0,C 180,E1 14182.462,E2 14182.462} C_VEL
LIN {X 0,Y 529.568,Z 934.937,A -85,B 0,C 180,E1 14187.003,E2 14187.003} C_VEL
LIN {X 0,Y 536.822,Z 892.112,A -85,B 0,C 180,E1 14188.955,E2 14188.955} C_VEL
LIN {X 0,Y 516.465,Z 847.917,A -85,B 0,C 180,E1 14195.066,E2 14195.066} C_VEL
LIN {X 0,Y 492.295,Z 810.992,A -85,B 0,C 180,E1 14202.846,E2 14202.846} C_VEL
LIN {X 0,Y 476.766,Z 789.876,A -85,B 0,C 180,E1 14210.019,E2 14210.019} C_VEL
LIN {X 0,Y 469.033,Z 781.4,A -85,B 0,C 180,E1 14216.041,E2 14216.041} C_VEL
LIN {X 0,Y 466.561,Z 778.77,A -85,B 0,C 180,E1 14225.812,E2 14225.812} C_VEL
LIN {X 0,Y 472.329,Z 785.618,A -85,B 0,C 180,E1 14232.854,E2 14232.854} C_VEL
LIN {X 0,Y 483.916,Z 800.481,A -85,B 0,C 180,E1 14239.554,E2 14239.554} C_VEL
LIN {X 0,Y 506.42,Z 831.253,A -85,B 0,C 180,E1 14247.643,E2 14247.643} C_VEL
LIN {X 0,Y 530.194,Z 874.324,A -85,B 0,C 180,E1 14254.513,E2 14254.513} C_VEL
LIN {X 0,Y 538.259,Z 896.726,A -85,B 0,C 180,E1 14257.075,E2 14257.075} C_VEL
LIN {X 0,Y 524.068,Z 965.288,A -85,B 0,C 180,E1 14260.149,E2 14260.149} C_VEL
LIN {X 0,Y 505.711,Z 1032.583,A -85,B 0,C 180,E1 14265.021,E2 14265.021} C_VEL
LIN {X 0,Y 486.873,Z 1093.469,A -85,B 0,C 180,E1 14271.818,E2 14271.818} C_VEL
LIN {X 0,Y 471.579,Z 1144.107,A -85,B 0,C 180,E1 14280.366,E2 14280.366} C_VEL
LIN {X 0,Y 462.929,Z 1178.968,A -85,B 0,C 180,E1 14289.367,E2 14289.367} C_VEL
LIN {X 0,Y 459.637,Z 1198.915,A -85,B 0,C 180,E1 14297.614,E2 14297.614} C_VEL
LIN {X 0,Y 459.134,Z 1208.348,A -85,B 0,C 180,E1 14305.261,E2 14305.261} C_VEL
LIN {X 0,Y 458.875,Z 1209.63,A -85,B 0,C 180,E1 14311.81,E2 14311.81} C_VEL
LIN {X 0,Y 451.094,Z 1207.141,A -85,B 0,C 180,E1 14316.173,E2 14316.173} C_VEL
LIN {X 0,Y 452.878,Z 1193.069,A -85,B 0,C 180,E1 14325.535,E2 14325.535} C_VEL
LIN {X 0,Y 458.882,Z 1163.929,A -85,B 0,C 180,E1 14335.439,E2 14335.439} C_VEL
LIN {X 0,Y 471.06,Z 1121.29,A -85,B 0,C 180,E1 14344.483,E2 14344.483} C_VEL
LIN {X 0,Y 488.691,Z 1065.79,A -85,B 0,C 180,E1 14352.143,E2 14352.143} C_VEL
LIN {X 0,Y 507.535,Z 1000.574,A -85,B 0,C 180,E1 14358.04,E2 14358.04} C_VEL
LIN {X 0,Y 524.454,Z 927.482,A -85,B 0,C 180,E1 14362.18,E2 14362.18} C_VEL
LIN {X 0,Y 529.197,Z 895.633,A -85,B 0,C 180,E1 14363.525,E2 14363.525} C_VEL
LIN {X 0,Y 501.888,Z 840.904,A -85,B 0,C 180,E1 14370.419,E2 14370.419} C_VEL
LIN {X 0,Y 473.881,Z 799.873,A -85,B 0,C 180,E1 14377.995,E2 14377.995} C_VEL
LIN {X 0,Y 454.485,Z 774.224,A -85,B 0,C 180,E1 14385.277,E2 14385.277} C_VEL
LIN {X 0,Y 450.263,Z 767.06,A -85,B 0,C 180,E1 14387.872,E2 14387.872} C_VEL
LIN {X 0,Y 451.025,Z 767.06,A -85,B 0,C 180,E1 14397.128,E2 14397.128} C_VEL
LIN {X 0,Y 450.556,Z 767.06,A -85,B 0,C 180,E1 14406.858,E2 14406.858} C_VEL
LIN {X 0,Y 449.904,Z 767.06,A -85,B 0,C 180,E1 14416.673,E2 14416.673} C_VEL
LIN {X 0,Y 450.125,Z 769.326,A -85,B 0,C 180,E1 14418.692,E2 14418.692} C_VEL
LIN {X 0,Y 463.215,Z 786.468,A -85,B 0,C 180,E1 14424.505,E2 14424.505} C_VEL
LIN {X 0,Y 486.635,Z 818.034,A -85,B 0,C 180,E1 14431.822,E2 14431.822} C_VEL
LIN {X 0,Y 515.185,Z 866.576,A -85,B 0,C 180,E1 14439.204,E2 14439.204} C_VEL
LIN {X 0,Y 528.446,Z 899.486,A -85,B 0,C 180,E1 14442.969,E2 14442.969} C_VEL
LIN {X 0,Y 512.948,Z 973.493,A -85,B 0,C 180,E1 14446.641,E2 14446.641} C_VEL
LIN {X 0,Y 494.33,Z 1040.479,A -85,B 0,C 180,E1 14452.018,E2 14452.018} C_VEL
LIN {X 0,Y 475.839,Z 1098.314,A -85,B 0,C 180,E1 14459.156,E2 14459.156} C_VEL
LIN {X 0,Y 461.672,Z 1144.064,A -85,B 0,C 180,E1 14467.809,E2 14467.809} C_VEL
LIN {X 0,Y 454.036,Z 1176.484,A -85,B 0,C 180,E1 14477.464,E2 14477.464} C_VEL
LIN {X 0,Y 451.344,Z 1194.623,A -85,B 0,C 180,E1 14487.114,E2 14487.114} C_VEL
LIN {X 0,Y 450.831,Z 1199.877,A -85,B 0,C 180,E1 14494.827,E2 14494.827} C_VEL
LIN {X 0,Y 451.204,Z 1196.061,A -85,B 0,C 180,E1 14503.61,E2 14503.61} C_VEL
LIN {X 0,Y 453.214,Z 1180.13,A -85,B 0,C 180,E1 14512.967,E2 14512.967} C_VEL
LIN {X 0,Y 459.485,Z 1151.521,A -85,B 0,C 180,E1 14522.266,E2 14522.266} C_VEL
LIN {X 0,Y 473.142,Z 1107.41,A -85,B 0,C 180,E1 14531.367,E2 14531.367} C_VEL
LIN {X 0,Y 492.096,Z 1050.675,A -85,B 0,C 180,E1 14539.029,E2 14539.029} C_VEL
LIN {X 0,Y 511.619,Z 987.269,A -85,B 0,C 180,E1 14544.602,E2 14544.602} C_VEL
LIN {X 0,Y 528.98,Z 914.854,A -85,B 0,C 180,E1 14548.634,E2 14548.634} C_VEL
LIN {X 0,Y 531.802,Z 896.427,A -85,B 0,C 180,E1 14549.464,E2 14549.464} C_VEL
LIN {X 0,Y 512.259,Z 853.149,A -85,B 0,C 180,E1 14555.65,E2 14555.65} C_VEL
LIN {X 0,Y 489.849,Z 817.925,A -85,B 0,C 180,E1 14563.279,E2 14563.279} C_VEL
LIN {X 0,Y 475.192,Z 797.589,A -85,B 0,C 180,E1 14570.334,E2 14570.334} C_VEL
LIN {X 0,Y 467.562,Z 788.863,A -85,B 0,C 180,E1 14576.61,E2 14576.61} C_VEL
LIN {X 0,Y 465.583,Z 786.754,A -85,B 0,C 180,E1 14585.825,E2 14585.825} C_VEL
LIN {X 0,Y 471.2,Z 793.636,A -85,B 0,C 180,E1 14592.767,E2 14592.767} C_VEL
LIN {X 0,Y 482.932,Z 809.039,A -85,B 0,C 180,E1 14599.599,E2 14599.599} C_VEL
LIN {X 0,Y 504.138,Z 839.158,A -85,B 0,C 180,E1 14607.474,E2 14607.474} C_VEL
LIN {X 0,Y 526.488,Z 881.294,A -85,B 0,C 180,E1 14614.286,E2 14614.286} C_VEL
LIN {X 0,Y 532.831,Z 900.904,A -85,B 0,C 180,E1 14616.507,E2 14616.507} C_VEL
LIN {X 0,Y 518.048,Z 969.232,A -85,B 0,C 180,E1 14619.664,E2 14619.664} C_VEL
LIN {X 0,Y 498.35,Z 1037.91,A -85,B 0,C 180,E1 14624.812,E2 14624.812} C_VEL
LIN {X 0,Y 478.739,Z 1098.202,A -85,B 0,C 180,E1 14631.85,E2 14631.85} C_VEL
LIN {X 0,Y 463.566,Z 1146.329,A -85,B 0,C 180,E1 14640.353,E2 14640.353} C_VEL
LIN {X 0,Y 454.861,Z 1180.45,A -85,B 0,C 180,E1 14649.506,E2 14649.506} C_VEL
LIN {X 0,Y 451.575,Z 1200.407,A -85,B 0,C 180,E1 14658.373,E2 14658.373} C_VEL
LIN {X 0,Y 451.241,Z 1209.312,A -85,B 0,C 180,E1 14667.108,E2 14667.108} C_VEL
LIN {X 0,Y 451.094,Z 1207.141,A -85,B 0,C 180,E1 14676.173,E2 14676.173} C_VEL
LIN {X 0,Y 443.595,Z 1202.243,A -85,B 0,C 180,E1 14680.591,E2 14680.591} C_VEL
LIN {X 0,Y 446.431,Z 1183.11,A -85,B 0,C 180,E1 14689.855,E2 14689.855} C_VEL
LIN {X 0,Y 454.909,Z 1150.087,A -85,B 0,C 180,E1 14699.301,E2 14699.301} C_VEL
LIN {X 0,Y 470.007,Z 1102.874,A -85,B 0,C 180,E1 14707.979,E2 14707.979} C_VEL
LIN {X 0,Y 489.349,Z 1043.389,A -85,B 0,C 180,E1 14715.112,E2 14715.112} C_VEL
LIN {X 0,Y 508.387,Z 976.277,A -85,B 0,C 180,E1 14720.306,E2 14720.306} C_VEL
LIN {X 0,Y 523.866,Z 900.039,A -85,B 0,C 180,E1 14723.995,E2 14723.995} C_VEL
LIN {X 0,Y 497.924,Z 846.441,A -85,B 0,C 180,E1 14730.919,E2 14730.919} C_VEL
LIN {X 0,Y 469.406,Z 803.519,A -85,B 0,C 180,E1 14739.074,E2 14739.074} C_VEL
LIN {X 0,Y 451.215,Z 780.662,A -85,B 0,C 180,E1 14746.285,E2 14746.285} C_VEL
LIN {X 0,Y 445.47,Z 773.409,A -85,B 0,C 180,E1 14749.474,E2 14749.474} C_VEL
LIN {X 0,Y 442.259,Z 767.06,A -85,B 0,C 180,E1 14752.134,E2 14752.134} C_VEL
LIN {X 0,Y 442.536,Z 767.06,A -85,B 0,C 180,E1 14761.002,E2 14761.002} C_VEL
LIN {X 0,Y 442.27,Z 767.06,A -85,B 0,C 180,E1 14770.893,E2 14770.893} C_VEL
LIN {X 0,Y 442.354,Z 769.209,A -85,B 0,C 180,E1 14774.479,E2 14774.479} C_VEL
LIN {X 0,Y 454.479,Z 784.508,A -85,B 0,C 180,E1 14781.349,E2 14781.349} C_VEL
LIN {X 0,Y 475.982,Z 813.471,A -85,B 0,C 180,E1 14789.155,E2 14789.155} C_VEL
LIN {X 0,Y 502.964,Z 857.008,A -85,B 0,C 180,E1 14796.714,E2 14796.714} C_VEL
LIN {X 0,Y 523.135,Z 901.16,A -85,B 0,C 180,E1 14802.341,E2 14802.341} C_VEL
LIN {X 0,Y 507.078,Z 975.1,A -85,B 0,C 180,E1 14806.058,E2 14806.058} C_VEL
LIN {X 0,Y 487.909,Z 1041.695,A -85,B 0,C 180,E1 14811.478,E2 14811.478} C_VEL
LIN {X 0,Y 468.807,Z 1099.312,A -85,B 0,C 180,E1 14818.703,E2 14818.703} C_VEL
LIN {X 0,Y 454.181,Z 1144.609,A -85,B 0,C 180,E1 14827.423,E2 14827.423} C_VEL
LIN {X 0,Y 446.151,Z 1176.865,A -85,B 0,C 180,E1 14837.239,E2 14837.239} C_VEL
LIN {X 0,Y 443.388,Z 1194.841,A -85,B 0,C 180,E1 14847.062,E2 14847.062} C_VEL
LIN {X 0,Y 442.833,Z 1199.983,A -85,B 0,C 180,E1 14854.914,E2 14854.914} C_VEL
LIN {X 0,Y 443.235,Z 1196.039,A -85,B 0,C 180,E1 14863.86,E2 14863.86} C_VEL
LIN {X 0,Y 445.363,Z 1179.953,A -85,B 0,C 180,E1 14873.396,E2 14873.396} C_VEL
LIN {X 0,Y 452.048,Z 1151.509,A -85,B 0,C 180,E1 14882.764,E2 14882.764} C_VEL
LIN {X 0,Y 466.51,Z 1107.268,A -85,B 0,C 180,E1 14892.023,E2 14892.023} C_VEL
LIN {X 0,Y 486.049,Z 1051.169,A -85,B 0,C 180,E1 14899.68,E2 14899.68} C_VEL
LIN {X 0,Y 506.24,Z 988.089,A -85,B 0,C 180,E1 14905.269,E2 14905.269} C_VEL
LIN {X 0,Y 524.302,Z 915.137,A -85,B 0,C 180,E1 14909.351,E2 14909.351} C_VEL
LIN {X 0,Y 526.294,Z 899.265,A -85,B 0,C 180,E1 14910.168,E2 14910.168} C_VEL
LIN {X 0,Y 507.158,Z 856.365,A -85,B 0,C 180,E1 14916.573,E2 14916.573} C_VEL
LIN {X 0,Y 484.209,Z 819.524,A -85,B 0,C 180,E1 14925.12,E2 14925.12} C_VEL
LIN {X 0,Y 472.366,Z 804.328,A -85,B 0,C 180,E1 14931.44,E2 14931.44} C_VEL
LIN {X 0,Y 466.489,Z 796.742,A -85,B 0,C 180,E1 14936.719,E2 14936.719} C_VEL
LIN {X 0,Y 464.626,Z 794.77,A -85,B 0,C 180,E1 14945.895,E2 14945.895} C_VEL
LIN {X 0,Y 470.076,Z 801.635,A -85,B 0,C 180,E1 14952.68,E2 14952.68} C_VEL
LIN {X 0,Y 482.549,Z 818.3,A -85,B 0,C 180,E1 14959.962,E2 14959.962} C_VEL
LIN {X 0,Y 503.547,Z 849.778,A -85,B 0,C 180,E1 14967.876,E2 14967.876} C_VEL
LIN {X 0,Y 524.262,Z 891.84,A -85,B 0,C 180,E1 14974.522,E2 14974.522} C_VEL
